(* CODESYS project tc3_utilities_extension.library
   Author: Csaba Attila Biro
   Placeholder: Tc3_Utilities_Extension
   Title: Tc3_Utilities_Extension
   Version: 2.4.92
   Company: Harman

Project tree, tasks and I/O mapping:
  libraries: Tc2_EtherCAT, * (Beckhoff Automation GmbH); Tc2_IoFunctions, * (Beckhoff Automation GmbH); Tc2_Standard, * (Beckhoff Automation GmbH); Tc2_System, * (Beckhoff Automation GmbH); Tc2_TcpIp, * (Beckhoff Automation GmbH); Tc2_Utilities, * (Beckhoff Automation GmbH); Tc3_EventLogger, * (Beckhoff Automation GmbH); Tc3_JsonXml, * (Beckhoff Automation GmbH); Tc3_Module, * (Beckhoff Automation GmbH)
  ConfigManager/
    function block FB_ConfigManager [ST]: FB_CALL_ACT, CREATE_PATH, Load, Save
  DataManager/
    JSON/
      function ANY_TO_JSON [ST]
      function CFG_TO_JSON [ST]
      global variables JSON_GVL
      function JSON_TO_ANY [ST]
      function JSON_TO_CFG [ST]
  EtherCatDiagnostic/
    DUTs/
      data type E_EcatDiagState
      data type E_EcCommState
      data type ST_EcMasterDevState
      data type ST_PortAddr
      data type ST_SlaveState
      data type ST_SlaveStateInfo
      data type ST_SlaveStateInfoScanned
      data type ST_TopologyData
    GVLs/
      global variables DIAG_GVL
    function block FB_EtherCATDiag [ST]: DiagnosticJson, M_CheckMasterDevState, M_GetScannedSlaveName, M_GetSlaveAdresses, M_GetSlaveIdentity, M_GetSlaveName, M_GetSlaveStates, M_GetTopoData, M_GetTopoDataLen, M_ScanSlaves
    function block FB_EtherCATDiagnosticWrapper [ST]
    function block FB_EtherCATFrameDiag [ST]
    function block FB_EtherCATSlaveInfo [ST]: M_GetScannedSlaveName, M_GetSlaveAdresses, M_GetSlaveIdentity, M_GetSlaveName, M_GetSlaveStates, M_GetTopoData, M_GetTopoDataLen, M_ScanSlaves
  EventLogger/
    DUTs/
      data type E_SubSystem
    global variables EVENT_GVL
    function block FB_EventHandler [ST]
    function block FB_EventLogger [ST]
  RecipeManager/
    function block FB_RecipeManager [ST]: ENUM_FILE_LIST_ACT, FB_CALL_ACT, CREATE_PATH, Load, RefreshNameList, Save, ValidateRecipe
  Tcp Barcode Reader/
    function block FB_BARCODE_READER [ST]: FB_CALL_ACT, READ, READ_REF
  TcpIpClients/
    DUTs/
      data type ENUM_DATA_EXCHANGE_STATE
    GVLs/
      global variables TCP_GVL
    function block FB_TCP_IP_CLIENT [ST]: FB_CALL_ACT, SEND
    function block FB_TCP_IP_CLIENT_LDAT [ST]: FB_CALL_ACT, SEND
  Test/
    DUTs/
      data type E_Task
      data type E_TaskState
      data type ST_Recipe
      data type ST_RecipeTask
    TASKs/
    program MAIN [ST]: FB_CALL_ACT
  TextFileHandlers/
    function block FB_ReadTextFile [ST]: Read
    function block FB_WriteTextFile [ST]: Write
    global variables FILE_GVL
  Version/
    global variables Global_Version
*)

// EtherCatDiagnostic/DUTs/E_EcatDiagState
{attribute 'to_string'}
TYPE E_EcatDiagState :
(
	Idle := 0,
    GetSlaveAddresses := 1,
    GetSlaveStates := 2,
    GetTopoDataLen := 3,
    GetTopoData := 4,
    ScanSlaves := 5,
    GetSlaveIdentity := 6,
    GetSlaveName := 7,
    GetScannedSlaveName := 8,
    LogDiagnostics := 9,
    Done := 8000
);
END_TYPE

// EtherCatDiagnostic/DUTs/E_EcCommState
TYPE E_EcCommState : (
	eEcState_UNDEFINED 	:= 0,
	eEcState_INIT 		:= 1,
	eEcState_PREOP 		:= 2,
	eEcState_BOOT 		:= 3,
	eEcState_SAFEOP 	:= 4,
	eEcState_OP 		:= 8
) UDINT;
END_TYPE

// EtherCatDiagnostic/DUTs/ST_EcMasterDevState
{attribute 'to_string'}
TYPE ST_EcMasterDevState :
STRUCT
	eEcState	 		: E_EcCommState;
	nReserved			: ARRAY [0..2] OF UINT;

	bLinkError			: BOOL;
	bResetRequired		: BOOL;
	bMissFrmRedMode		: BOOL;
	bWatchdogTriggerd	: BOOL;
	bDriverNotFound		: BOOL;
	bResetActive		: BOOL;
	bAtLeastOneNotInOp	: BOOL;
	bDcNotInSync		: BOOL;
END_STRUCT
END_TYPE

// EtherCatDiagnostic/DUTs/ST_PortAddr
{attribute 'to_string'}
TYPE ST_PortAddr :
STRUCT
	portA : UINT;
	portB : UINT;
	portC : UINT;
	portD : UINT;
END_STRUCT
END_TYPE

// EtherCatDiagnostic/DUTs/ST_SlaveState
{attribute 'to_string'}
TYPE ST_SlaveState :
STRUCT
	(* slave state *)
	eEcState 		: E_EcCommState;
	nReserved		: UINT;
	bError			: BOOL;
	bInvalidVPRS	: BOOL;
	nReserved2		: UINT;

	(* link state *)
	bNoCommToSlave	: BOOL;
	bLinkError		: BOOL;
	bMissingLink	: BOOL;
	bUnexpectedLink	: BOOL;
	bPortA			: BOOL;
	bPortB			: BOOL;
	bPortC			: BOOL;
	bPortD			: BOOL;
END_STRUCT
END_TYPE

// EtherCatDiagnostic/DUTs/ST_SlaveStateInfo
{attribute 'to_string'}
TYPE ST_SlaveStateInfo :
STRUCT
	nIndex 			: DINT;
	sName 			: STRING(255); 		(* name of slave given in System Manager *)
	sType 			: STRING(255);		(* type of slave, e.g. EK1100*)
	nECAddr 		: UINT;			(* EtherCAT Slave Addr *)
	bDiagData		: BOOL;			(* DiagData in Slave State *)
	stPortCRCErrors	: ST_EcCrcErrorEx;(* Slave CRC-Errors, separate for each Port *)
	nSumCRCErrors	: UDINT;		(* Slave CRC-Errors, sum of all Ports *)
	stState 		: ST_SlaveState;(* EtherCAT State and Link state*)
END_STRUCT
END_TYPE

// EtherCatDiagnostic/DUTs/ST_SlaveStateInfoScanned
{attribute 'to_string'}
TYPE ST_SlaveStateInfoScanned :
STRUCT
	nIndex 			: DINT;
	sName 			: STRING; 		(* name of slave given in System Manager *)
	sType 			: STRING;		(* type of slave, e.g. EK1100*)
	nECAddr 		: UINT;			(* EtherCAT Slave Addr *)
	bDifferentName	: BOOL;			(* Name of Scanned configuration differs from Configured configuration *)
	bDifferentType	: BOOL;			(* Type Of Scanned configuration differs from Configured configuration *)
	bDifferentAddr	: BOOL;			(* EcAddress of Scanned configuration differs from Configured configuration *)
END_STRUCT
END_TYPE

// EtherCatDiagnostic/DUTs/ST_TopologyData
{attribute 'to_string'}
TYPE ST_TopologyData :
STRUCT
	iOwnPhysicalAddr 	: UINT;
	iOwnAutoIncAddr		: UINT;
	stPhysicalAddr		: ST_PortAddr;
	stAutoIncAddr		: ST_PortAddr;
	iPortDelay			: ARRAY [0..2] OF UDINT; (* EC_AD, EC_DB, EC_BC *)
	iReserved			: ARRAY [0..7] OF UDINT;
END_STRUCT
END_TYPE

// EventLogger/DUTs/E_SubSystem
TYPE E_SubSystem :
(
	NILVALUE := 0,
	SAFETY := 1,
	LOGIC := 2,
	MOTION := 3,
	FIELDBUS := 4,
	PNEUMATIC := 5,
	ELECTRIC := 6
)WORD;
END_TYPE

// TcpIpClients/DUTs/ENUM_DATA_EXCHANGE_STATE
TYPE ENUM_DATA_EXCHANGE_STATE :
(
	E_IDLE := 0,
	E_SEND_START := 100,
	E_SEND_WAIT := 200,
	E_RECEIVE_START := 300,
	E_RECEIVE_WAIT := 400,
	E_DONE := 2000,
	
	E_ERROR:=15000		
);
END_TYPE

// Test/DUTs/E_Task
TYPE E_Task :
(
	TASK_START:=0,
	TASK_MOVE,
	TASK_TAKE_SCREW,
	TASK_SCREWING,
	TASK_BARCODE_SCANN,
	TASK_CAMERA_CHECK,
	TASK_ADAPTER,
	TASK_END
	
(*
	TASK_START:= 			'EMPTY'
	TASK_MOVE:=				'X:=-86.36;Y:=168.56;Z:=115.23;C:=90.12;'
	TASK_TAKE_SCREW:=		'X:=-86.36;Y:=168.56;Z:=115.23;C:=90.12;FEEDER:=2;'
	TASK_SCREWING:=			'PRE_SCREWING:=111;MAIN_SCREWING:=11;DEPTH_TARGET:=5.89;DEPTH_REF:=11.96;'
	TASK_BARCODE_SCANN:=	'IP_ADDRESS:=192.168.0.51;'
	TASK_CAMERA_CHECK:=		'PRG_ID:=192.168.0.51;',
	TASK_ADAPTER:=			'ADAPTER_TASK_ID:=2;',
	TASK_END:= 				'EMPTY'
*)

);
END_TYPE

// Test/DUTs/E_TaskState
TYPE E_TaskState :
(
	TASK_READY:=0,
	TASK_BUSY,
	TASK_DONE,
	TASK_OK,
	TASK_NG
);
END_TYPE

// Test/DUTs/ST_Recipe
TYPE ST_Recipe :
STRUCT
	DESCRIPTION:		STRING(100);
	RECIPE_LOADED:		BOOL;
	TASK_LIST:			ARRAY [1..500] OF ST_RecipeTask;	
END_STRUCT
END_TYPE

// Test/DUTs/ST_RecipeTask
TYPE ST_RecipeTask :
STRUCT
	SLOT_CHANGE:			BOOL:=FALSE;	(* Change slot after finished this position TASK *)	
	TASK:					E_Task;		(* Describe what we want to do in *)
	TASK_COMMENT:			STRING;
	TASK_PARAMETER:			STRING(255);
	
	(*
		TASK_START:= 			'EMPTY'
		TASK_MOVE:=				'X:=-86.36;Y:=168.56;Z:=115.23;C:=90.12;'
		TASK_TAKE_SCREW:=		'X:=-86.36;Y:=168.56;Z:=115.23;C:=90.12;FEEDER:=2;'
		TASK_SCREWING:=			'PRE_SCREWING:=111;MAIN_SCREWING:=11;DEPTH_TARGET:=5.89;DEPTH_REF:=11.96;'
		TASK_BARCODE_SCANN:=	'IP_ADDRESS:=192.168.0.51;'
		TASK_CAMERA_CHECK:=		'PRG_ID:=192.168.0.51;',
		TASK_ADAPTER:=			'ADAPTER_TASK_ID:=2;',
		TASK_END:= 				'EMPTY'
	*)
	
	TASK_RESULT:			E_TaskState;
END_STRUCT
END_TYPE

// DataManager/JSON/JSON_GVL
VAR_GLOBAL CONSTANT
	MAX_JSON_LENGTH:UDINT:=1000000; //1MB - 0.001GB
	CFG_JSON_LENGTH:UDINT:=15000;
END_VAR

// EtherCatDiagnostic/GVLs/DIAG_GVL
VAR_GLOBAL CONSTANT
	iSLAVEADDR_ARR_SIZE	: UINT := 256;
    ESC_MAX_PORTS : UINT := 3;
END_VAR

// EventLogger/EVENT_GVL
{attribute 'qualified_only'}
VAR_GLOBAL
	G_bAlarmActive:			BOOL;
	G_sAlarmMessage:		STRING(255);
	G_sAlarmSource:			STRING(255);
	G_sAlarmJson:			STRING(7000);
END_VAR

// TcpIpClients/GVLs/TCP_GVL
VAR_GLOBAL CONSTANT
	DEFAULT_TIMEOUT:								TIME:=T#5S;
	DEFAULT_RECONNECT:								TIME:=T#1S;
	DEFAULT_SDAT_LENGTH:							UDINT:=998;
	DEFAULT_LDAT_LENGTH:							UDINT:=49998;
	DEFAULT_STX:									BYTE:=16#02;
	DEFAULT_ETX:									BYTE:=16#03;
END_VAR

// TextFileHandlers/FILE_GVL
VAR_GLOBAL CONSTANT
	MAX_FILE_LENGTH:UDINT:=1000000; //1MB - 0.001GB
END_VAR

// Version/Global_Version
{attribute 'TcGenerated'}
{attribute 'no-analysis'}
{attribute 'linkalways'}
// This function has been automatically generated from the project information.
VAR_GLOBAL CONSTANT
	{attribute 'const_non_replaced'}
	stLibVersion_Tc3_Utilities_Extension : ST_LibVersion := (iMajor := 2, iMinor := 4, iBuild := 92, iRevision := 0, nFlags := 0, sVersion := '2.4.92');
END_VAR

// ConfigManager/FB_ConfigManager
FUNCTION_BLOCK FB_ConfigManager
VAR_INPUT
	sDef:				STRING(MAX_STRING_LENGTH):='Configuration';
	sExt:				STRING(MAX_STRING_LENGTH):='cfg';
	sFolderPath:		STRING(MAX_STRING_LENGTH):='C:\TwinCAT\Tc_Data\Configuration';
	sKey:				STRING(MAX_STRING_LENGTH):='Configuration';
	pData:				PVOID;
	nData:				UDINT;
	RESET:				BOOL;
END_VAR
VAR_OUTPUT
	READY:				BOOL;
	BUSY:				BOOL;
	DONE:				BOOL;
	
	ERROR:				BOOL;
	ERROR_ID:			UDINT;
	
	TIME_STAMP:			STRING(MAX_STRING_LENGTH);
END_VAR
VAR
	FB_SYSTIME: 		FB_LocalSystemTime:= (bEnable:= TRUE, dwCycle:= 1);
	WRITE_FILE:			FB_WriteTextFile;
	READ_FILE:			FB_ReadTextFile;
	
	JSON_STRING:		STRING(CFG_JSON_LENGTH);
	JSON_LENGTH:		UDINT;
	
	STATE:				INT;
	INIT:				BOOL:=TRUE;
	EXECUTE:			BOOL;
	
	FILE_PATH:			STRING(MAX_STRING_LENGTH);
	FILE_NAME:			STRING(MAX_STRING_LENGTH);
	RECIPE_NAME:		STRING(MAX_STRING_LENGTH):='DefaultName';
	
	FB_CreateDir: 			FB_CreateDir;
	FB_FIND_FILE: 			FB_EnumFindFileEntry:= (sNetID:= '', tTimeout:= DEFAULT_ADS_TIMEOUT);
	ENUM_FIND_FILE:			STRING(MAX_STRING_LENGTH);
	ENUM_FIND_RECIPENAME:	STRING;
	ENUM_INDEX:				UDINT:=1;
	ENUMERATE: 				BOOL;
	ENUM_STATE: 			INT;
	
	eSubSystem: 			E_SubSystem:= E_SubSystem.LOGIC;
	FB_LOGGER:				FB_EventLogger:= (eSubsystem:= eSubsystem, sJson:='{}');
END_VAR

CREATE_PATH();
FB_FIND_FILE(sPathName:= CONCAT(sFolderPath, CONCAT('\', CONCAT('*', CONCAT('.', CONCAT(sDef, CONCAT('.', sExt)))))));
FB_SYSTIME();
READY:= STATE=0;
BUSY:= STATE<>0;

IF INIT THEN
	INIT := FALSE;
	ENUMERATE:=TRUE;
    FB_CreateDir( bExecute := FALSE );
    FB_CreateDir(sNetId:= '',
                sPathName:= sFolderPath,
                ePath:= PATH_GENERIC,
                bExecute:= TRUE,
                tTimeout:= DEFAULT_ADS_TIMEOUT);
ELSE
    FB_CreateDir(bExecute := FALSE);
END_IF

CASE STATE OF
	1100:
		ENUMERATE:=TRUE;
		CREATE_PATH();
		IF CFG_TO_JSON(pData,nData, sKey:=sKey, SYSTEMTIME_TO_STRING(FB_SYSTIME.systemTime), JSON_STRING, JSON_LENGTH) THEN
			STATE:=1200;
		END_IF
	1200:
		IF WRITE_FILE.Write(FILE_PATH) THEN
			STATE:=1300;
		END_IF
	2100:
		CREATE_PATH();
		IF READ_FILE.Read(FILE_PATH) THEN
			STATE:=2200;
		END_IF
	2200:
		IF JSON_TO_CFG(pData,nData, sKey:=sKey, TIME_STAMP, JSON_STRING) THEN
			EXECUTE:=FALSE;
			ENUMERATE:=TRUE;
			STATE:=2300;
		END_IF
END_CASE

ERROR:=(ERROR_ID<>0);
FB_CALL_ACT();

ACTION FB_CALL_ACT:
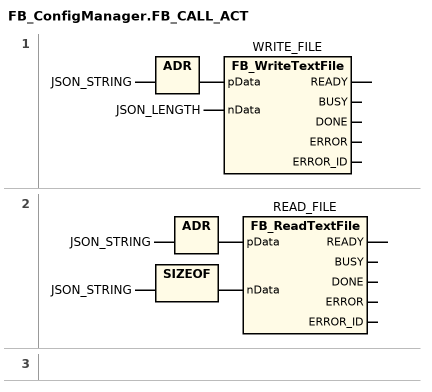
// NETWORK 1
WRITE_FILE(pData := ADR(JSON_STRING), nData := JSON_LENGTH); // FB_WriteTextFile

// NETWORK 2
READ_FILE(pData := ADR(JSON_STRING), nData := SIZEOF(JSON_STRING)); // FB_ReadTextFile

// NETWORK 3
END_ACTION

METHOD PRIVATE CREATE_PATH : BOOL
VAR_INPUT
END_VAR
FILE_NAME:=CONCAT(RECIPE_NAME, CONCAT('.', CONCAT(sDef, CONCAT('.', sExt))));
FILE_PATH:=CONCAT(sFolderPath, CONCAT('\', FILE_NAME));
END_METHOD

METHOD PUBLIC Load : BOOL
VAR_INPUT
	NAME:				STRING;
END_VAR
VAR
END_VAR
IF STATE=0 THEN
	RECIPE_NAME:=NAME;
	STATE:=2100;
END_IF

IF STATE=2300 THEN
	STATE:=0;
	Load:=TRUE;
	RETURN;
END_IF
END_METHOD

METHOD PUBLIC Save : BOOL
VAR_INPUT
	NAME:				STRING;
END_VAR
VAR
END_VAR
IF STATE=0 THEN
	RECIPE_NAME:=NAME;
	STATE:=1100;
END_IF
IF STATE=1300 THEN
	STATE:=0;
	Save:=TRUE;
	RETURN;
END_IF
END_METHOD

END_FUNCTION_BLOCK

// DataManager/JSON/CFG_TO_JSON
(*
	Convert any type to JSON string
*)
FUNCTION CFG_TO_JSON : BOOL
VAR_INPUT
	pData:					PVOID;
	nData:					UDINT;
	sKey:					STRING;
	sTimeStamp:				STRING;
	sJson:					REFERENCE TO STRING(CFG_JSON_LENGTH);
	cbJson:					REFERENCE TO UDINT;
END_VAR
VAR
	sDataType: 				STRING;
	REF_VALID:				BOOL;
	JSON_WRITER: 			FB_JsonSaxWriter;
  	JSON_DATA: 				FB_JsonReadWriteDataType;
	eSubSystem: 			E_SubSystem:= E_SubSystem.LOGIC;
	FB_LOGGER:				FB_EventLogger:= (eSubsystem:= eSubsystem);
END_VAR

REF_VALID:=(__ISVALIDREF(sJson) AND __ISVALIDREF(cbJson) AND (pData<>0 AND nData>0));

IF REF_VALID THEN
	sDataType:=JSON_DATA.GetDataTypeNameByAddress(nData:=nData, pData:=pData);
	MEMSET(ADR(sJson), 0, SIZEOF(sJson));
	JSON_WRITER.ResetDocument();
	JSON_WRITER.StartObject();
	JSON_WRITER.AddKeyString('Timestamp', sTimeStamp);
	JSON_DATA.AddJsonKeyValueFromSymbol(fbWriter:=JSON_WRITER, sKey:=sKey, sDatatype:=sDataType, nData:=nData, pData:=pData);
	JSON_WRITER.EndObject();
	cbJson:=JSON_WRITER.CopyDocument(sJson, SIZEOF(sJson));
	CFG_TO_JSON:=TRUE;
ELSE
	IF pData=0 THEN
		FB_LOGGER(sMsg:='Check data pointer failed due to invalid destination address.', eSevr:=TcEventSeverity.Error);
	ELSIF nData<=0 THEN
		FB_LOGGER(sMsg:='Check data pointer failed due to invalid size.', eSevr:=TcEventSeverity.Error);
	ELSIF NOT __ISVALIDREF(sJson) THEN
		FB_LOGGER(sMsg:='Check JSON string failed due to invalid reference.', eSevr:=TcEventSeverity.Error);
	ELSIF NOT __ISVALIDREF(cbJson) THEN
		FB_LOGGER(sMsg:='Check JSON length failed due to invalid reference.', eSevr:=TcEventSeverity.Error);
	END_IF
	CFG_TO_JSON:=TRUE;
END_IF

END_FUNCTION

// EventLogger/FB_EventLogger
{attribute 'reflection'}
FUNCTION_BLOCK FB_EventLogger
VAR_INPUT
	sMsg			: T_MaxString;
	eSevr			: TcEventSeverity	:= TcEventSeverity.Verbose;
	eSubSystem		: E_SubSystem;
	sJson			: STRING(7000)	:= '{}';
END_VAR

VAR_OUTPUT
END_VAR

VAR
	bInitialized		:	BOOL := FALSE;
	bInitFailed			:	BOOL := FALSE;
	sSubsystemSource	:	STRING;
	fbMessage			:	REFERENCE TO FB_TcMessage;
	fbAlarm				:	REFERENCE TO FB_TcAlarm;
	fbMessages 			:	ARRAY [0..4] OF FB_TcMessage;
	fbAlarms			:	ARRAY [0..4] OF FB_TcAlarm;
	fbSource 			:	FB_TcSourceInfo;
	hr 					:	HRESULT;
	hrLastInternalError :	HRESULT;
	eTraceLevel 		:	TcEventSeverity := TcEventSeverity.Verbose;
	
	{attribute 'instance-path'} 
    {attribute 'noinit'} 
	sPath				:	T_MaxString;
END_VAR

IF NOT bInitialized AND NOT bInitFailed THEN
	//Messages
	hr := fbMessages[TC_EVENTS.GeneralEventClass.Verbose.nEventId].CreateEx(TC_EVENTS.GeneralEventClass.Verbose, 0);
	IF FAILED(hr) THEN
		bInitFailed := TRUE;
		hrLastInternalError := hr;
	END_IF
	hr := fbMessages[TC_EVENTS.GeneralEventClass.Info.nEventId].CreateEx(TC_EVENTS.GeneralEventClass.Info, 0);
	IF FAILED(hr) THEN
		bInitFailed := TRUE;
		hrLastInternalError := hr;
	END_IF
	hr := fbMessages[TC_EVENTS.GeneralEventClass.Warning.nEventId].CreateEx(TC_EVENTS.GeneralEventClass.Warning, 0);
	IF FAILED(hr) THEN
		bInitFailed := TRUE;
		hrLastInternalError := hr;
	END_IF
	//Alarm messages
	hr := fbMessages[TC_EVENTS.GeneralEventClass.Error.nEventId].CreateEx(TC_EVENTS.GeneralEventClass.Error, 0);
	IF FAILED(hr) THEN
		bInitFailed := TRUE;
		hrLastInternalError := hr;
	END_IF
	hr := fbMessages[TC_EVENTS.GeneralEventClass.Critical.nEventId].CreateEx(TC_EVENTS.GeneralEventClass.Critical, 0);
	IF FAILED(hr) THEN
		bInitFailed := TRUE;
		hrLastInternalError := hr;
	END_IF	
	//Alarms
	hr := fbAlarms[TC_EVENTS.GeneralEventClass.Error.nEventId].CreateEx(TC_EVENTS.GeneralEventClass.Error, TRUE, 0);
	IF FAILED(hr) THEN
		bInitFailed := TRUE;
		hrLastInternalError := hr;
	END_IF
	hr := fbAlarms[TC_EVENTS.GeneralEventClass.Critical.nEventId].CreateEx(TC_EVENTS.GeneralEventClass.Critical, TRUE, 0);
	IF FAILED(hr) THEN
		bInitFailed := TRUE;
		hrLastInternalError := hr;
	END_IF	
	
	//Init failed
	IF bInitFailed THEN
		ADSLOGSTR(msgCtrlMask := ADSLOG_MSGTYPE_ERROR, msgFmtStr:='[LOGGER] Initialization failed in %s', strArg:=sPath); 
	ELSE
		bInitialized := TRUE;
	END_IF
END_IF
IF bInitFailed THEN
	RETURN;
END_IF
CASE eSevr OF
	//Messages
	TcEventSeverity.Verbose: 	fbMessage REF= fbMessages[TC_EVENTS.GeneralEventClass.Verbose.nEventId];
	TcEventSeverity.Info:		fbMessage REF= fbMessages[TC_EVENTS.GeneralEventClass.Info.nEventId];	
	TcEventSeverity.Warning:	fbMessage REF= fbMessages[TC_EVENTS.GeneralEventClass.Warning.nEventId];
	//Alarms
	TcEventSeverity.Error:		
		fbMessage REF= fbMessages[TC_EVENTS.GeneralEventClass.Error.nEventId]; 
		fbAlarm REF= fbAlarms[TC_EVENTS.GeneralEventClass.Error.nEventId]; 
	TcEventSeverity.Critical:	
		fbMessage REF= fbMessages[TC_EVENTS.GeneralEventClass.Critical.nEventId];
		fbAlarm REF= fbAlarms[TC_EVENTS.GeneralEventClass.Critical.nEventId];
	ELSE
		RETURN;
END_CASE
CASE eSubsystem OF
	E_Subsystem.FIELDBUS: sSubsystemSource := ' - EtherCAT';
	E_Subsystem.MOTION: sSubsystemSource := ' - Motion';
	E_Subsystem.SAFETY: sSubsystemSource := ' - Safety';
	E_Subsystem.LOGIC: sSubsystemSource := ' - Logic';
	E_Subsystem.PNEUMATIC: sSubsystemSource := ' - Pneumatic';	
	E_Subsystem.ELECTRIC: sSubsystemSource := ' - Electric';	
	ELSE
		sSubsystemSource := 'Unknown';
END_CASE
sMsg:=CONCAT(' ',CONCAT(sMsg,' '));
IF eSevr=TcEventSeverity.Verbose OR eSevr=TcEventSeverity.Info OR eSevr=TcEventSeverity.Warning THEN
	fbSource.sName :=CONCAT(sPath, sSubsystemSource);
	hr := fbMessage.CreateEx(stEventEntry:=fbMessage.stEventEntry, ipSourceInfo:=fbSource);
	fbMessage.ipArguments.Clear();
	fbMessage.ipArguments.AddString(sMsg);
	IF LEN(sJson) = 0 THEN
		sJson := '{}';
	END_IF
	fbMessage.SetJsonAttribute(sJson);
	IF NOT FAILED(hr) AND fbMessage.eSeverity >= eTraceLevel THEN
		hr := fbMessage.Send(0);
	END_IF
	IF FAILED(hr) THEN
		hrLastInternalError := hr;
	END_IF
ELSIF eSevr=TcEventSeverity.Error OR eSevr=TcEventSeverity.Critical THEN
	fbSource.sName :=CONCAT(sPath, sSubsystemSource);
	hr := fbAlarm.CreateEx(stEventEntry:=fbAlarm.stEventEntry, ipSourceInfo:=fbSource, bWithConfirmation:=TRUE);
	fbAlarm.ipArguments.Clear();
	
	fbAlarm.ipArguments.AddString(sMsg);
	IF LEN(sJson) = 0 THEN
		sJson := '{}';
	END_IF
	fbAlarm.SetJsonAttribute(sJson);
	IF NOT FAILED(hr) AND fbAlarm.eSeverity >= eTraceLevel THEN
		hr := fbAlarm.Raise(0);
		EVENT_GVL.G_sAlarmJson:=sJson;
		EVENT_GVL.G_sAlarmSource:=fbSource.sName;
		EVENT_GVL.G_sAlarmMessage:=sMsg;
		EVENT_GVL.G_bAlarmActive:=TRUE;
	END_IF
	IF FAILED(hr) THEN
		hrLastInternalError := hr;
	END_IF
	hr := fbMessage.CreateEx(stEventEntry:=fbMessage.stEventEntry, ipSourceInfo:=fbSource);
	fbMessage.ipArguments.Clear();
	fbMessage.ipArguments.AddString(sMsg);
	IF LEN(sJson) = 0 THEN
		sJson := '{}';
	END_IF
	fbMessage.SetJsonAttribute(sJson);
	IF NOT FAILED(hr) AND fbMessage.eSeverity >= eTraceLevel THEN
		hr := fbMessage.Send(0);
	END_IF
	IF FAILED(hr) THEN
		hrLastInternalError := hr;
	END_IF
END_IF

END_FUNCTION_BLOCK

// DataManager/JSON/JSON_TO_CFG
(*
	Convert JSON string to any sutitable type
*)
FUNCTION JSON_TO_CFG : BOOL
VAR_INPUT
	pData:					PVOID;
	nData:					UDINT;
	sKey:					STRING;
	sTimeStamp:				REFERENCE TO STRING;
	sJson:					REFERENCE TO STRING(CFG_JSON_LENGTH);
END_VAR
VAR
	sDataType: 				STRING;
	sDataSymbol:			STRING;
	REF_VALID:				BOOL;
	JSON_DOM_PARSER: 		FB_JsonDomParser;
	JSON_DOC: 				SJsonValue;
	JSON_TIME: 				SJsonValue;
	JSON_CONTENT:			SJsonValue;
  	JSON_DATA: 				FB_JsonReadWriteDataType;
	eSubSystem: 			E_SubSystem:= E_SubSystem.LOGIC;
	FB_LOGGER:				FB_EventLogger:= (eSubsystem:= eSubsystem);
END_VAR

REF_VALID:=(__ISVALIDREF(sJson) AND __ISVALIDREF(sTimeStamp) AND (pData<>0 AND nData>0));

IF REF_VALID THEN
	sDataType:=JSON_DATA.GetDataTypeNameByAddress(nData:=nData, pData:=pData);
	sDataSymbol:=JSON_DATA.GetSymbolNameByAddress(nData:=nData, pData:=pData);
	
	JSON_DOC:=JSON_DOM_PARSER.ParseDocument(sJson);
	IF JSON_DOM_PARSER.HasMember(JSON_DOC, 'Timestamp') THEN
		JSON_TIME:=JSON_DOM_PARSER.FindMember(JSON_DOC, 'Timestamp');
		sTimeStamp:=JSON_DOM_PARSER.GetString(JSON_TIME);
	END_IF
	IF JSON_DOM_PARSER.HasMember(JSON_DOC, sKey) THEN
		MEMSET(ADR(sJson), 0, SIZEOF(sJson));
		JSON_CONTENT:=JSON_DOM_PARSER.FindMember(JSON_DOC, sKey);
		JSON_DOM_PARSER.CopyJson (JSON_CONTENT, sJson, SIZEOF(sJson));
		JSON_DATA.SetSymbolFromJson(sJson:=sJson, sDatatype:=sDataType, nData:=nData, pData:=pData);
	END_IF
	JSON_TO_CFG:=TRUE;
ELSE
	IF pData=0 THEN
		FB_LOGGER(sMsg:='Check data pointer failed due to invalid destination address.', eSevr:=TcEventSeverity.Error);
	ELSIF nData<=0 THEN
		FB_LOGGER(sMsg:='Check data pointer failed due to invalid size.', eSevr:=TcEventSeverity.Error);
	ELSIF NOT __ISVALIDREF(sJson) THEN
		FB_LOGGER(sMsg:='Check JSON string failed due to invalid reference.', eSevr:=TcEventSeverity.Error);
	ELSIF NOT __ISVALIDREF(sTimeStamp) THEN
		FB_LOGGER(sMsg:='Check TimeStamp string failed due to invalid reference.', eSevr:=TcEventSeverity.Error);
	END_IF
	JSON_TO_CFG:=TRUE;
END_IF

END_FUNCTION

// TextFileHandlers/FB_WriteTextFile
{attribute 'reflection'}
FUNCTION_BLOCK FB_WriteTextFile
VAR_INPUT
	pData:				PVOID;
	nData:				UDINT;
END_VAR
VAR_OUTPUT
	READY:				BOOL;
	BUSY:				BOOL;
	DONE:				BOOL;
	ERROR:				BOOL;
	ERROR_ID:			UDINT;
END_VAR
VAR
	FB_FileWrite:		FB_FileWrite;
	FB_FileOpen:		FB_FileOpen;
	FB_FileClose:		FB_FileClose;
	sPath:				STRING(MAX_STRING_LENGTH);
	H_DEST_FILE:		UINT:= 0;
	STATE:				INT;
	EXECUTE:			BOOL;
	
	eSubSystem: 			E_SubSystem:= E_SubSystem.LOGIC;
	FB_LOGGER:				FB_EventLogger:= (eSubsystem:= eSubsystem);
END_VAR

READY:= STATE=0;
BUSY:= STATE<>0;
CASE STATE OF
	0:
		IF EXECUTE THEN
			ERROR_ID:=0;
			DONE:=FALSE;
			STATE:=100;
		END_IF
	100:
		FB_FileOpen( bExecute := FALSE );
		FB_FileOpen( sNetId := '', sPathName := sPath,
					 nMode := FOPEN_MODEWRITE OR FOPEN_MODETEXT,
					 ePath := PATH_GENERIC, tTimeout := DEFAULT_ADS_TIMEOUT, bExecute := TRUE );
		STATE:=200;
    200:
		FB_FileOpen( bExecute := FALSE );
		IF NOT FB_FileOpen.bBusy THEN
			IF FB_FileOpen.bError THEN
				ERROR_ID:=FB_FileOpen.nErrId;
				FB_LOGGER(sMsg:=CONCAT('FB_FileOpen throw an error: ', DWORD_TO_HEXSTR(ERROR_ID, 0, FALSE )), eSevr:=TcEventSeverity.Error);
				STATE:=700;
			ELSE
				H_DEST_FILE := FB_FileOpen.hFile;
				STATE:=300;
			END_IF
		END_IF
	300:
		FB_FileWrite( bExecute := FALSE );
        FB_FileWrite( sNetId:='', 
					  hFile:=H_DEST_FILE,
                      pWriteBuff:= pData, 
					  cbWriteLen:= (nData-1),
                      bExecute:=TRUE, 
					  tTimeout:=DEFAULT_ADS_TIMEOUT );
		STATE:=400;
	400:
		FB_FileWrite( bExecute := FALSE );
		IF NOT FB_FileWrite.bBusy THEN
			IF FB_FileWrite.bError THEN
				ERROR_ID:=FB_FileWrite.nErrId;
				FB_LOGGER(sMsg:=CONCAT('FB_FileWrite throw an error: ', DWORD_TO_HEXSTR(ERROR_ID, 0, FALSE )), eSevr:=TcEventSeverity.Error);
				STATE:=700;
			ELSE
				STATE:=500;
			END_IF
		END_IF
	 500:
         FB_FileClose( bExecute := FALSE );
         FB_FileClose( sNetId:='', hFile:=H_DEST_FILE, bExecute:=TRUE, tTimeout:=DEFAULT_ADS_TIMEOUT );
         STATE:=600;
     600:
		FB_FileClose( bExecute := FALSE );
		IF NOT FB_FileClose.bBusy THEN
			IF FB_FileClose.bError THEN
				ERROR_ID:=FB_FileClose.nErrId;
				FB_LOGGER(sMsg:=CONCAT('FB_FileClose throw an error: ', DWORD_TO_HEXSTR(ERROR_ID, 0, FALSE )), eSevr:=TcEventSeverity.Error);
			END_IF
			STATE:=700;
			DONE:=TRUE;
			H_DEST_FILE:= 0;
		END_IF
	700:
		IF NOT EXECUTE THEN
			STATE:=0;
		END_IF
END_CASE

METHOD PUBLIC Write : BOOL
VAR_INPUT
	sFilePath:		STRING(MAX_STRING_LENGTH);
END_VAR
IF sFilePath<>'' THEN
	IF STATE=700 THEN
		EXECUTE:=FALSE;
		Write:=TRUE;
	END_IF
	
	IF STATE=0 THEN
		sPath:=sFilePath;
		EXECUTE:=TRUE;
	END_IF	
END_IF
END_METHOD

END_FUNCTION_BLOCK

// TextFileHandlers/FB_ReadTextFile
{attribute 'reflection'}
FUNCTION_BLOCK FB_ReadTextFile
VAR_INPUT
	pData:				PVOID;
	nData:				UDINT;
END_VAR
VAR_OUTPUT
	READY:				BOOL;
	BUSY:				BOOL;
	DONE:				BOOL;
	ERROR:				BOOL;
	ERROR_ID:			UDINT;
END_VAR
VAR
	FB_FileRead:		FB_FileRead;
	FB_FileOpen:		FB_FileOpen;
	FB_FileClose:		FB_FileClose;
	sPath:				STRING(MAX_STRING_LENGTH);
	H_SCR_FILE:			UINT:= 0;
	STATE:				INT;
	EXECUTE:			BOOL;
	
	eSubSystem: 			E_SubSystem:= E_SubSystem.LOGIC;
	FB_LOGGER:				FB_EventLogger:= (eSubsystem:= eSubsystem);
END_VAR

READY:= STATE=0;
BUSY:= STATE<>0;
CASE STATE OF
	0:
		IF EXECUTE THEN
			ERROR_ID:=0;
			DONE:=FALSE;
			MEMSET(pData, 0, nData);
			STATE:=100;
		END_IF
	100:	
		FB_FileOpen( bExecute := FALSE );
		FB_FileOpen( sNetId := '', sPathName := sPath,
					 nMode := FOPEN_MODEREAD OR FOPEN_MODETEXT,
					 ePath := PATH_GENERIC, tTimeout := DEFAULT_ADS_TIMEOUT, bExecute := TRUE );
		STATE:=200;
	200:
		FB_FileOpen( bExecute := FALSE );
		IF NOT FB_FileOpen.bBusy THEN
			IF FB_FileOpen.bError THEN
				ERROR_ID:=FB_FileOpen.nErrId;
				FB_LOGGER(sMsg:=CONCAT(CONCAT('FB_FileOpen throw an error: ', DWORD_TO_HEXSTR(ERROR_ID, 0, FALSE )),CONCAT(' Path: ', sPath)), eSevr:=TcEventSeverity.Error);
				STATE:=700;
			ELSE
				H_SCR_FILE := FB_FileOpen.hFile;
				STATE:=300;
			END_IF
		END_IF
	300:
		FB_FileRead( bExecute:= FALSE );
		FB_FileRead( sNetId:='', hFile:=H_SCR_FILE,
					pReadBuff:= pData, cbReadLen:= nData,
					bExecute:=TRUE, tTimeout:=DEFAULT_ADS_TIMEOUT);
		STATE:=400;
	400:
		FB_FileRead( bExecute:= FALSE );
		IF NOT FB_FileRead.bBusy THEN
			IF FB_FileRead.bError THEN
				ERROR_ID:=FB_FileRead.nErrId;
				FB_LOGGER(sMsg:=CONCAT('FB_FileRead throw an error: ', DWORD_TO_HEXSTR(ERROR_ID, 0, FALSE )), eSevr:=TcEventSeverity.Error);
				STATE:=700;
			ELSE
				STATE:=500;
			END_IF
		END_IF
	500:
         FB_FileClose( bExecute := FALSE );
         FB_FileClose( sNetId:='', hFile:=H_SCR_FILE, bExecute:=TRUE, tTimeout:=DEFAULT_ADS_TIMEOUT );
         STATE:=600;
	600:
		FB_FileClose( bExecute := FALSE );
		IF NOT FB_FileClose.bBusy THEN
			IF FB_FileClose.bError THEN
				ERROR_ID:=FB_FileClose.nErrId;
				FB_LOGGER(sMsg:=CONCAT('FB_FileClose throw an error: ', DWORD_TO_HEXSTR(ERROR_ID, 0, FALSE )), eSevr:=TcEventSeverity.Error);
			END_IF
			STATE:=700;
			DONE:=TRUE;
			H_SCR_FILE := 0;
		END_IF
	700:
		IF NOT EXECUTE THEN
			STATE:=0;
		END_IF
END_CASE

ERROR:=(ERROR_ID<>0);

METHOD PUBLIC Read : BOOL
VAR_INPUT
	sFilePath:		STRING(MAX_STRING_LENGTH);
END_VAR
IF sFilePath<>'' THEN
	IF STATE=700 THEN
		EXECUTE:=FALSE;
		Read:=TRUE;
	END_IF
	
	IF STATE=0 THEN
		sPath:=sFilePath;
		EXECUTE:=TRUE;
	END_IF
END_IF
END_METHOD

END_FUNCTION_BLOCK

// DataManager/JSON/ANY_TO_JSON
(*
	Convert any type to JSON string
*)
FUNCTION ANY_TO_JSON : BOOL
VAR_INPUT
	pData:					PVOID;
	nData:					UDINT;
	sKey:					STRING;
	sTimeStamp:				STRING;
	sJson:					REFERENCE TO STRING(MAX_JSON_LENGTH);
	cbJson:					REFERENCE TO UDINT;
END_VAR
VAR
	sDataType: 				STRING;
	REF_VALID:				BOOL;
	JSON_WRITER: 			FB_JsonSaxWriter;
  	JSON_DATA: 				FB_JsonReadWriteDataType;
	eSubSystem: 			E_SubSystem:= E_SubSystem.LOGIC;
	FB_LOGGER:				FB_EventLogger:= (eSubsystem:= eSubsystem);
END_VAR

REF_VALID:=(__ISVALIDREF(sJson) AND __ISVALIDREF(cbJson) AND (pData<>0 AND nData>0));

IF REF_VALID THEN
	sDataType:=JSON_DATA.GetDataTypeNameByAddress(nData:=nData, pData:=pData);
	MEMSET(ADR(sJson), 0, SIZEOF(sJson));
	JSON_WRITER.ResetDocument();
	JSON_WRITER.StartObject();
	JSON_WRITER.AddKeyString('Timestamp', sTimeStamp);
	JSON_DATA.AddJsonKeyValueFromSymbol(fbWriter:=JSON_WRITER, sKey:=sKey, sDatatype:=sDataType, nData:=nData, pData:=pData);
	JSON_WRITER.EndObject();
	cbJson:=JSON_WRITER.CopyDocument(sJson, SIZEOF(sJson));
	ANY_TO_JSON:=TRUE;
ELSE
	IF pData=0 THEN
		FB_LOGGER(sMsg:='Check data pointer failed due to invalid destination address.', eSevr:=TcEventSeverity.Error);
	ELSIF nData<=0 THEN
		FB_LOGGER(sMsg:='Check data pointer failed due to invalid size.', eSevr:=TcEventSeverity.Error);
	ELSIF NOT __ISVALIDREF(sJson) THEN
		FB_LOGGER(sMsg:='Check JSON string failed due to invalid reference.', eSevr:=TcEventSeverity.Error);
	ELSIF NOT __ISVALIDREF(cbJson) THEN
		FB_LOGGER(sMsg:='Check JSON length failed due to invalid reference.', eSevr:=TcEventSeverity.Error);
	END_IF
	ANY_TO_JSON:=TRUE;
END_IF

END_FUNCTION

// DataManager/JSON/JSON_TO_ANY
(*
	Convert JSON string to any sutitable type
*)
FUNCTION JSON_TO_ANY : BOOL
VAR_INPUT
	pData:					PVOID;
	nData:					UDINT;
	sKey:					STRING;
	sTimeStamp:				REFERENCE TO STRING;
	sJson:					REFERENCE TO STRING(MAX_JSON_LENGTH);
END_VAR
VAR
	sDataType: 				STRING;
	sDataSymbol:			STRING;
	REF_VALID:				BOOL;
	JSON_DOM_PARSER: 		FB_JsonDomParser;
	JSON_DOC: 				SJsonValue;
	JSON_TIME: 				SJsonValue;
	JSON_CONTENT:			SJsonValue;
  	JSON_DATA: 				FB_JsonReadWriteDataType;
	eSubSystem: 			E_SubSystem:= E_SubSystem.LOGIC;
	FB_LOGGER:				FB_EventLogger:= (eSubsystem:= eSubsystem);
END_VAR

REF_VALID:=(__ISVALIDREF(sJson) AND __ISVALIDREF(sTimeStamp) AND (pData<>0 AND nData>0));

IF REF_VALID THEN
	sDataType:=JSON_DATA.GetDataTypeNameByAddress(nData:=nData, pData:=pData);
	sDataSymbol:=JSON_DATA.GetSymbolNameByAddress(nData:=nData, pData:=pData);
	JSON_DOC:=JSON_DOM_PARSER.ParseDocument(sJson);
	IF JSON_DOM_PARSER.HasMember(JSON_DOC, 'Timestamp') THEN
		JSON_TIME:=JSON_DOM_PARSER.FindMember(JSON_DOC, 'Timestamp');
		sTimeStamp:=JSON_DOM_PARSER.GetString(JSON_TIME);
	END_IF
	IF JSON_DOM_PARSER.HasMember(JSON_DOC, sKey) THEN
		MEMSET(ADR(sJson), 0, SIZEOF(sJson));
		JSON_CONTENT:=JSON_DOM_PARSER.FindMember(JSON_DOC, sKey);
		JSON_DOM_PARSER.CopyJson (JSON_CONTENT, sJson, SIZEOF(sJson));
		JSON_DATA.SetSymbolFromJson(sJson:=sJson, sDatatype:=sDataType, nData:=nData, pData:=pData);
	END_IF
	JSON_TO_ANY:=TRUE;
ELSE
	IF pData=0 THEN
		FB_LOGGER(sMsg:='Check data pointer failed due to invalid destination address.', eSevr:=TcEventSeverity.Error);
	ELSIF nData<=0 THEN
		FB_LOGGER(sMsg:='Check data pointer failed due to invalid size.', eSevr:=TcEventSeverity.Error);
	ELSIF NOT __ISVALIDREF(sJson) THEN
		FB_LOGGER(sMsg:='Check JSON string failed due to invalid reference.', eSevr:=TcEventSeverity.Error);
	ELSIF NOT __ISVALIDREF(sTimeStamp) THEN
		FB_LOGGER(sMsg:='Check TimeStamp string failed due to invalid reference.', eSevr:=TcEventSeverity.Error);
	END_IF
	JSON_TO_ANY:=TRUE;
END_IF

END_FUNCTION

// EtherCatDiagnostic/FB_EtherCATDiag
FUNCTION_BLOCK FB_EtherCATDiag
VAR_INPUT
	sIPCNetID					: T_AmsNetId; 	// AmsNetId of the IPC 
	sMasterNetID				: T_AmsNetId; 	// AmsNetId of the EtherCAT master device 
	nMasterDevID				: UINT;			// Device ID of EtherCAT master
	nSlaveCount 				: UINT;			// current slave count
	nSlaveCountCfg 				: UINT;			// configured slave count
	nMasterDevState				: WORD;			// device state of EtherCAT Master
	bAllFrameWcStatesOK			: BOOL;			// all FrameWcState OK?
	tTimeout					: TIME := T#5S; // ads timeout
    eSubSystem 					: E_SubSystem := E_SubSystem.FIELDBUS;
END_VAR
VAR_OUTPUT
	bEtherCATOK					: BOOL;			// no problem on EtherCAT
	bFrameWcStateError			: BOOL;			// error in at least one frame
	bSlaveCountError			: BOOL;			// EtherCAT slave count mismatch (# of cfg slaves <> # of found slaves)
	bMasterDevStateError		: BOOL;			// error in master device state
	stMasterDevState			: ST_EcMasterDevState; // splitted master device state
	bBusy						: BOOL;			// FB busy
	bError						: BOOL;			// FB with error
	iErrorID					: UDINT;		// FB error ID
END_VAR
VAR_IN_OUT
	arrDiagSlaveInfo 			: ARRAY [0..ESC_MAX_PORTS] OF ST_SlaveStateInfo;		// read in info from configured slaves
	arrDiagSlaveInfoScanned		: ARRAY [0..ESC_MAX_PORTS] OF ST_SlaveStateInfoScanned;	// read in info from scanned slaves
END_VAR
VAR
	sMasterOpState				: STRING(255);
	sSlaveOpState				: STRING(255);
	iState						: E_EcatDiagState;
	nMasterDevStatePrev			: WORD;
	bSlaveCountErrorPrev		: BOOL;
	bAllFrameWcStatesOKPrev		: BOOL;
	bDiagReq					: BOOL := TRUE;
	I							: UDINT;
    P							: UDINT;   
    arrSlaveInfo 				: ARRAY [0..iSLAVEADDR_ARR_SIZE] OF ST_SlaveStateInfo;
    rSlaveInfo  				: REFERENCE TO ST_SlaveStateInfo;

	(* -- Get Slave Addresses *)
	fbGetSlaveAddresses 		: FB_EcGetAllSlaveAddr;
	arrSlaveAddresses 			: ARRAY[0..iSLAVEADDR_ARR_SIZE] OF UINT;
	iNumOfSlavesRead			: UINT;

	(* -- Get Slave States *)
	fbGetAllSlaveStates			: FB_EcGetAllSlaveStates;
	arrSlaveStates 				: ARRAY[0..iSLAVEADDR_ARR_SIZE] OF ST_EcSlaveState;

	(* -- Get Topology Data *)
	iTopologyData				: UDINT;
	fbGetTopologyData			: ADSREAD;
	arrTopologyData				: ARRAY[0..iSLAVEADDR_ARR_SIZE] OF ST_TopologyData;

	(* -- Check Topology *)
	aiDiagIndex					: ARRAY [0..ESC_MAX_PORTS] OF UINT;
    iDiagIndex 					: UINT;    
	aiDiagPort					: ARRAY [0..ESC_MAX_PORTS] OF UINT;
    iDiagPort 					: UINT;
	iIdx						: DINT;

	(* -- Scan Slaves *)
	fbEcGetScannedSlaves		: FB_EcGetScannedSlaves;
	arrScannedSlaveInfo			: ARRAY [0..iSLAVEADDR_ARR_SIZE] OF ST_EcSlaveScannedData; // what...
    rScannedSlaveInfo   		: REFERENCE TO ST_EcSlaveScannedData;
	nScannedSlaves				: UINT;

	(* -- Get Slave Identities *)
	fbGetSlaveIdentity			: FB_EcGetSlaveIdentity;
	stIdentity 					: ST_EcSlaveIdentity;

	(* -- Get Slave Names *)
	fbGetSlaveName 				: IOF_GetBoxNameByAddr;
    arrSlaveInfoScanned			: ARRAY [0..iSLAVEADDR_ARR_SIZE] OF ST_SlaveStateInfoScanned; // the F
    rSlaveInfoScanned   		: REFERENCE TO ST_SlaveStateInfoScanned;
	strName						: STRING;

    // Logging components
    fbLogger 					: FB_EventLogger := (eSubsystem := eSubsystem);  
    fbJson 						: FB_JsonSaxWriter;
    fbJsonDataType 				: FB_JsonReadWriteDataType;
    rDiagSlaveInfo 				: REFERENCE TO ST_SlaveStateInfo;
    tEtherCATOK 				: F_TRIG;
    tFrameWcStateError 			: R_TRIG;
    tMasterError 				: R_TRIG;
    jsonIdx 					: UINT;
    test 						: T_MaxString;
END_VAR


(* cyclic diag *)
bFrameWcStateError := NOT bAllFrameWcStatesOK;

bSlaveCountError := (nSlaveCount <> nSlaveCountCfg) OR (nSlaveCount = 0);
IF (bSlaveCountError AND NOT bSlaveCountErrorPrev) OR (NOT bSlaveCountError AND bSlaveCountErrorPrev) THEN
	bSlaveCountErrorPrev := bSlaveCountError;
	bDiagReq := TRUE; // slave count error change detected --> diag required
END_IF

IF (bAllFrameWcStatesOK AND NOT bAllFrameWcStatesOKPrev) OR (NOT bAllFrameWcStatesOK AND bAllFrameWcStatesOKPrev) THEN
	bAllFrameWcStatesOKPrev := bAllFrameWcStatesOK;
	bDiagReq := TRUE; // frame error change detected --> diag required
END_IF

IF (nMasterDevState <> nMasterDevStatePrev) THEN
	M_CheckMasterDevState();
	bDiagReq := TRUE; // devstate change detected --> diag required
END_IF

(* acyclic diag *)
CASE iState OF
E_EcatDiagState.Idle: (* IDLE *)
	IF bDiagReq THEN				// diag requested
		bDiagReq := FALSE;

		IF sMasterNetID <> '' AND sMasterNetID <> '0.0.0.0.0.0' THEN
			iState := E_EcatDiagState.GetSlaveAddresses;	// execute diag
			bBusy := TRUE;
		ELSE
			bError := TRUE;
			iErrorID := 7;
		END_IF

		bEtherCATOK := FALSE;
	ELSE
		// check for changes in idle
		IF (bSlaveCountError OR bMasterDevStateError OR NOT bAllFrameWcStatesOK) AND NOT (arrSlaveInfo[aiDiagIndex[0]].bDiagData) THEN
			bEtherCATOK := FALSE;
			bDiagReq := TRUE;//new error --> diag requested    
		ELSIF (bSlaveCountError AND NOT bSlaveCountErrorPrev) OR (NOT bSlaveCountError AND bSlaveCountErrorPrev) THEN
			bSlaveCountErrorPrev := bSlaveCountError;
			bEtherCATOK := FALSE;
			bDiagReq := TRUE;// slave count error change detected --> diag required
		ELSIF (nMasterDevState <> nMasterDevStatePrev) THEN
			bEtherCATOK := FALSE;
			bDiagReq := TRUE;// devstate change detected --> diag required
		ELSIF (bAllFrameWcStatesOK AND NOT bAllFrameWcStatesOKPrev) OR (NOT bAllFrameWcStatesOK AND bAllFrameWcStatesOKPrev) THEN
			bAllFrameWcStatesOKPrev := bAllFrameWcStatesOK;
			bEtherCATOK := FALSE;
			bDiagReq := TRUE;// frame error change detected --> diag required
		ELSIF (bSlaveCountError OR bMasterDevStateError OR NOT bAllFrameWcStatesOK OR arrSlaveInfo[aiDiagIndex[0]].bDiagData) THEN
			bEtherCATOK := FALSE;
		ELSE
			bEtherCATOK := TRUE;
		END_IF
	END_IF

E_EcatDiagState.GetSlaveAddresses: (* get adresses *)
	M_GetSlaveAdresses();

E_EcatDiagState.GetSlaveStates: (* get states *)
	M_GetSlaveStates();

E_EcatDiagState.GetTopoDataLen:	(* get topology data length *)
	M_GetTopoDataLen();

E_EcatDiagState.GetTopoData:	(* get topology data *)
	M_GetTopoData();

E_EcatDiagState.ScanSlaves:	(* scan slaves *)
	M_ScanSlaves();

E_EcatDiagState.GetSlaveIdentity:	(* get identity *)
	M_GetSlaveIdentity();

E_EcatDiagState.GetSlaveName:	(* get name *)
	M_GetSlaveName();

E_EcatDiagState.GetScannedSlaveName:	(* get scanned name *)
	M_GetScannedSlaveName();

E_EcatDiagState.LogDiagnostics: (* Log diagnostics *)
    IF jsonIdx < iNumOfSlavesRead THEN // the last entry is always blank
        jsonIdx := MIN(iSLAVEADDR_ARR_SIZE, jsonIdx);
        rDiagSlaveInfo REF= arrSlaveInfo[jsonIdx];
		DiagnosticJson();
		IF rDiagSlaveInfo.sName <> '' THEN
			fbLogger(sMsg:=CONCAT('EtherCAT diagnostic result of ', rDiagSlaveInfo.sName), eSevr:=TcEventSeverity.Info);
		END_IF
        jsonIdx := jsonIdx + 1;
    ELSE
        jsonIdx := 0;
        iState := E_EcatDiagState.Done;    
	END_IF   
    
E_EcatDiagState.Done:	(* DONE *)
	bBusy := FALSE;
	iState := 0;

END_CASE

// Log messages
tEtherCATOK(CLK:=bEtherCATOK);
IF tEtherCATOK.Q THEN
    fbLogger(sMsg:='EtherCAT failure detected, starting diagnostic sequnce', eSevr:=TcEventSeverity.Critical, sJson:='');
END_IF

tFrameWcStateError(CLK:=bFrameWcStateError);
IF tFrameWcStateError.Q THEN
    fbLogger(sMsg:='WorkingCounterFrame error in at least one frame.', eSevr:=TcEventSeverity.Error, sJson:='');
END_IF

tMasterError(CLK:=bMasterDevStateError);
IF tMasterError.Q THEN
	CASE stMasterDevState.eEcState OF
		0: sMasterOpState:= 'UNDEFINED';
		1: sMasterOpState:= 'INIT';
		2: sMasterOpState:= 'PREOP';
		3: sMasterOpState:= 'BOOT';
		4: sMasterOpState:= 'SAFEOP';
		8: sMasterOpState:= 'OP';
	END_CASE
    fbJson.StartObject();
        fbJson.AddKey('EtherCAT Master Diagnostic');
        fbJson.StartObject();
            fbJson.AddKey('At least one not in OP state');
            fbJson.AddBool(stMasterDevState.bAtLeastOneNotInOp);
            fbJson.AddKey('DC not in sync');
            fbJson.AddBool(stMasterDevState.bDcNotInSync);
            fbJson.AddKey('Driver not found');
            fbJson.AddBool(stMasterDevState.bDriverNotFound);
            fbJson.AddKey('Link error');
            fbJson.AddBool(stMasterDevState.bLinkError);
            fbJson.AddKey('Miss Frm red mode');
            fbJson.AddBool(stMasterDevState.bMissFrmRedMode);
            fbJson.AddKey('Reset active');
            fbJson.AddBool(stMasterDevState.bResetActive);
            fbJson.AddKey('Reset required');
            fbJson.AddBool(stMasterDevState.bResetRequired);
            fbJson.AddKey('Watchdog triggerd');
            fbJson.AddBool(stMasterDevState.bWatchdogTriggerd);
            fbJson.AddKey('EtherCAT-State');
            fbJson.AddString(sMasterOpState);
        fbJson.EndObject();
    fbJson.EndObject();
    fbJson.CopyDocument(fbLogger.sJson, SIZEOF(fbLogger.sJson));

    fbLogger(sMsg:=CONCAT('Error in EtherCAT Master device state. EtherCAT-State: ', sMasterOpState), eSevr:=TcEventSeverity.Critical);
    fbJson.ResetDocument();
END_IF

ACTION DiagnosticJson:
CASE rDiagSlaveInfo.stState.eEcState OF
	0: sSlaveOpState:= 'UNDEFINED';
	1: sSlaveOpState:= 'INIT';
	2: sSlaveOpState:= 'PREOP';
	3: sSlaveOpState:= 'BOOT';
	4: sSlaveOpState:= 'SAFEOP';
	8: sSlaveOpState:= 'OP';
END_CASE
fbJson.StartObject();
    fbJson.AddKey('EtherCAT Diagnostic');
    fbJson.StartObject();
        
        fbJson.AddKey('EtherCAT address');
        fbJson.AddUdint(rDiagSlaveInfo.nECAddr);
        
        fbJson.AddKey('Index');
        fbJson.AddDint(rDiagSlaveInfo.nIndex);
        
        fbJson.AddKey('Name');
        fbJson.AddString(rDiagSlaveInfo.sName);
        
        fbJson.AddKey('Type');
        fbJson.AddString(rDiagSlaveInfo.sType);
    
        fbJson.AddKey('Diagnostic data');
        fbJson.AddBool(rDiagSlaveInfo.bDiagData);
        
        fbJson.AddKey('EtherCAT port CRC errors');
        fbjson.StartObject();
        
            fbJson.AddKey('Port - A');
            fbJson.AddUdint(rDiagSlaveInfo.stPortCRCErrors.portA);
            fbJson.AddKey('Port - B');
            fbJson.AddUdint(rDiagSlaveInfo.stPortCRCErrors.portB);
            fbJson.AddKey('Port - C');
            fbJson.AddUdint(rDiagSlaveInfo.stPortCRCErrors.portC);
            fbJson.AddKey('Port - D');
            fbJson.AddUdint(rDiagSlaveInfo.stPortCRCErrors.portD);
            
        fbJson.EndObject();
        
        fbJson.AddKey('Summary of CRC errors');
        fbjson.AddUdint(rDiagSlaveInfo.nSumCRCErrors);
        
        fbJson.AddKey('Terminal state');
        fbJson.StartObject();
        
            fbJson.AddKey('EtherCAT-State');
            fbJson.AddString(sSlaveOpState);
//            fbJson.AddKey('Reserved 1');
//            fbJson.AddUdint(rDiagSlaveInfo.stState.nReserved);
            fbJson.AddKey('Error');
            fbJson.AddBool(rDiagSlaveInfo.stState.bError);
            fbJson.AddKey('Invalid VPRS');
            fbJson.AddBool(rDiagSlaveInfo.stState.bInvalidVPRS);
//            fbJson.AddKey('Reserved 2');
//            fbJson.AddUdint(rDiagSlaveInfo.stState.nReserved2);
            fbJson.AddKey('No communication to slave');
            fbJson.AddBool(rDiagSlaveInfo.stState.bNoCommToSlave);
            fbJson.AddKey('Link error');
            fbJson.AddBool(rDiagSlaveInfo.stState.bLinkError);
            fbJson.AddKey('Missing link');
            fbJson.AddBool(rDiagSlaveInfo.stState.bMissingLink);
            fbJson.AddKey('Unexpected link');
            fbJson.AddBool(rDiagSlaveInfo.stState.bUnexpectedLink);
            fbJson.AddKey('Port - A');
            fbJson.AddBool(rDiagSlaveInfo.stState.bPortA);
            fbJson.AddKey('Port - B');
            fbJson.AddBool(rDiagSlaveInfo.stState.bPortB);
            fbJson.AddKey('Port - C');
            fbJson.AddBool(rDiagSlaveInfo.stState.bPortC);
            fbJson.AddKey('Port - D');
            fbJson.AddBool(rDiagSlaveInfo.stState.bPortD);
    
        fbJson.EndObject();
    
    fbJson.EndObject();
    
fbJson.EndObject();

fbJson.CopyDocument(fbLogger.sJson, SIZEOF(fbLogger.sJson));
fbJson.ResetDocument();
END_ACTION

ACTION M_CheckMasterDevState:
(* check master errors based on devstate *)
bMasterDevStateError 				:= nMasterDevState <> 0;
stMasterDevState.bLinkError 		:= ((nMasterDevState AND 16#000F) = 1) OR ((nMasterDevState AND 16#000F) = 4);
stMasterDevState.bResetRequired 	:= ((nMasterDevState AND 16#000F) = 2) OR ((nMasterDevState AND 16#FFF0) = 16#10);
stMasterDevState.bMissFrmRedMode 	:= (nMasterDevState AND 16#000F) = 8;
stMasterDevState.bWatchdogTriggerd 	:= (nMasterDevState AND 16#20) = 16#20;
stMasterDevState.bDriverNotFound 	:= (nMasterDevState AND 16#40) = 16#40;
stMasterDevState.bResetActive 		:= (nMasterDevState AND 16#80) = 16#80;
stMasterDevState.bAtLeastOneNotInOp := ((nMasterDevState AND 16#100) = 16#100) OR ((nMasterDevState AND 16#200) = 16#200) OR
										((nMasterDevState AND 16#400) = 16#400) OR ((nMasterDevState AND 16#800) = 16#800);
stMasterDevState.bDcNotInSync 		:= (nMasterDevState AND 16#1000) = 16#1000;
nMasterDevStatePrev 				:= nMasterDevState;
END_ACTION

ACTION M_GetScannedSlaveName:

rSlaveInfoScanned REF= arrSlaveInfoScanned[aiDiagIndex[iIdx]];
rScannedSlaveInfo REF= arrScannedSlaveInfo[aiDiagIndex[iIdx]];

fbGetSlaveName(
	NETID		:= sIPCNetId,
	DEVICEID	:= nMasterDevID,
	BOXADDR		:= rScannedSlaveInfo.nAddr,
	START		:= TRUE,
	TMOUT		:= tTimeout,
	BOXNAME		=> strName
);

IF NOT fbGetSlaveName.BUSY THEN
	fbGetSlaveName(START:= FALSE);

	(* add scanned info *)
	rSlaveInfoScanned.nIndex 	:= iDiagIndex + 1;
	IF rScannedSlaveInfo.nAddr <> 0 THEN
		IF NOT fbGetSlaveName.ERR THEN
			rSlaveInfoScanned.sName := strName;
		END_IF
	ELSE
		rSlaveInfoScanned.sType		:= '';
	END_IF

	IF (iDiagIndex < nScannedSlaves) THEN
		rSlaveInfoScanned.sType		:= F_ConvProductCodeToString(rScannedSlaveInfo.stSlaveIdentity);
	ELSE
		rSlaveInfoScanned.sType		:= '';
	END_IF

	rSlaveInfoScanned.nECAddr	:= rScannedSlaveInfo.nAddr;

	IF rSlaveInfoScanned.sName <> rSlaveInfo.sName THEN
		rSlaveInfoScanned.bDifferentName := TRUE;
	ELSE
		rSlaveInfoScanned.bDifferentName := FALSE;
	END_IF

	IF rSlaveInfoScanned.nECAddr <> rSlaveInfo.nECAddr THEN
		rSlaveInfoScanned.bDifferentAddr := TRUE;
	ELSE
		rSlaveInfoScanned.bDifferentAddr := FALSE;
	END_IF

	IF rSlaveInfoScanned.sType <> rSlaveInfo.sType THEN
		rSlaveInfoScanned.bDifferentType := TRUE;
	ELSE
		rSlaveInfoScanned.bDifferentType := FALSE;
	END_IF

	IF iIdx < ESC_MAX_PORTS THEN
		iIdx := iIdx + 1;
		iState := E_EcatDiagState.GetSlaveIdentity; // loop back
	ELSE
		iIdx := 0;
		iState := E_EcatDiagState.LogDiagnostics;

		FOR I := 0 TO ESC_MAX_PORTS DO
			IF aiDiagPort[I] <> 0 THEN
				arrDiagSlaveInfo[I] := arrSlaveInfo[aiDiagIndex[I]];
				arrDiagSlaveInfoScanned[I] := arrSlaveInfoScanned[aiDiagIndex[I]];
			ELSE
				MEMSET(ADR(arrDiagSlaveInfo[I]), 0, SIZEOF(arrDiagSlaveInfo[I]));
				MEMSET(ADR(arrDiagSlaveInfoScanned[I]), 0, SIZEOF(arrDiagSlaveInfoScanned[I]));
			END_IF
		END_FOR
	END_IF
END_IF
END_ACTION

ACTION M_GetSlaveAdresses:
fbGetSlaveAddresses(
	sNetId		:= sMasterNetID,
	pAddrBuf	:= ADR(arrSlaveAddresses),
	cbBufLen	:= SIZEOF(arrSlaveAddresses),
	bExecute	:= TRUE,
	tTimeout	:= tTimeout,
	nSlaves		=> iNumOfSlavesRead
);

IF NOT fbGetSlaveAddresses.bBusy THEN
	fbGetSlaveAddresses(bExecute:= FALSE);
	IF NOT fbGetSlaveAddresses.bError THEN
		FOR I := 0 TO MIN(iNumOfSlavesRead, iSLAVEADDR_ARR_SIZE) DO
			arrSlaveInfo[I].nECAddr := arrSlaveAddresses[I];
		END_FOR
	END_IF
	iState := GetSlaveStates;
END_IF
END_ACTION

ACTION M_GetSlaveIdentity:

iDiagIndex := aiDiagIndex[iIdx];
iDiagPort := aiDiagPort[iIdx];

rSlaveInfo REF= arrSlaveInfo[iDiagIndex];

fbGetSlaveIdentity(
	sNetId		:= sMasterNetID,
	nSlaveAddr	:= rSlaveInfo.nECAddr,
	bExecute	:= TRUE,
	tTimeout	:= tTimeout,
	identity	=> stIdentity
);

IF NOT fbGetSlaveIdentity.bBusy THEN
	fbGetSlaveIdentity(bExecute:= FALSE);

	IF NOT fbGetSlaveIdentity.bError THEN
		IF aiDiagPort[iIdx] <> 0 THEN
			rSlaveInfo.nIndex	:= aiDiagIndex[iIdx] + 1;
			rSlaveInfo.sType 	:= F_ConvProductCodeToString(stSlaveIdentity := stIdentity);
		END_IF
	END_IF
	iState := E_EcatDiagState.GetSlaveName;
END_IF
END_ACTION

ACTION M_GetSlaveName:
fbGetSlaveName(
	NETID		:= sIPCNetId,
	DEVICEID	:= nMasterDevID,
	BOXADDR		:= rSlaveInfo.nECAddr,
	START		:= TRUE,
	TMOUT		:= tTimeout,
	BOXNAME		=> strName
);

IF NOT fbGetSlaveName.BUSY THEN
	fbGetSlaveName(START:= FALSE);

	IF NOT fbGetSlaveName.ERR THEN
		IF iDiagPort <> 0 THEN
			rSlaveInfo.sName 	:= strName;
		END_IF
	END_IF

	iState := E_EcatDiagState.GetScannedSlaveName;
END_IF
END_ACTION

ACTION M_GetSlaveStates:
fbGetAllSlaveStates(
	sNetId		:= sMasterNetID,
	pStateBuf	:= ADR(arrSlaveStates),
	cbBufLen	:= SIZEOF(arrSlaveStates),
	bExecute	:= TRUE,
	tTimeout	:= tTimeout,
	nSlaves		=> iNumOfSlavesRead
);

IF NOT fbGetAllSlaveStates.bBusy THEN
	fbGetAllSlaveStates(bExecute:= FALSE);

	IF NOT fbGetAllSlaveStates.bError THEN
		IF iNumOfSlavesRead = nSlaveCountCfg THEN
			FOR I := 0 TO ESC_MAX_PORTS DO
				aiDiagIndex[I] := 0;
			END_FOR

			(* split slave state and link state *)
			FOR I := 0 TO MIN(iNumOfSlavesRead, iSLAVEADDR_ARR_SIZE) DO
				(* slave state*)
				arrSlaveInfo[I].stState.eEcState 		:= arrSlaveStates[I].deviceState AND 16#0F;
				arrSlaveInfo[I].stState.bError 			:= arrSlaveStates[I].deviceState.4;
				arrSlaveInfo[I].stState.bInvalidVPRS 	:= arrSlaveStates[I].deviceState.5;
				(* link state *)
				arrSlaveInfo[I].stState.bNoCommToSlave 	:= arrSlaveStates[I].linkState.0;
				arrSlaveInfo[I].stState.bLinkError 		:= arrSlaveStates[I].linkState.1;
				arrSlaveInfo[I].stState.bMissingLink 	:= arrSlaveStates[I].linkState.2;
				arrSlaveInfo[I].stState.bUnexpectedLink := arrSlaveStates[I].linkState.3;
				arrSlaveInfo[I].stState.bPortA 			:= arrSlaveStates[I].linkState.4;
				arrSlaveInfo[I].stState.bPortB 			:= arrSlaveStates[I].linkState.5;
				arrSlaveInfo[I].stState.bPortC 			:= arrSlaveStates[I].linkState.6;
				arrSlaveInfo[I].stState.bPortD 			:= arrSlaveStates[I].linkState.7;
				(* DiagData *)
				arrSlaveInfo[I].bDiagData	:= ((arrSlaveStates[I].deviceState AND 16#F0) <> 0) OR
					(((arrSlaveStates[I].deviceState AND 16#0F) > 0) AND ((arrSlaveStates[I].deviceState AND 16#0F) < 8)) OR
					(arrSlaveStates[I].linkState <> 0);

				IF arrSlaveInfo[I].bDiagData THEN
					IF (I=0) THEN
						aiDiagIndex[0] := 0;
					ELSE
						IF (aiDiagIndex[0] = 0) AND NOT arrSlaveInfo[0].bDiagData THEN
							aiDiagIndex[0] :=  UDINT_TO_UINT(I);
						END_IF
					END_IF
				END_IF
			END_FOR
		END_IF
	END_IF

	IF arrSlaveInfo[aiDiagIndex[0]].bDiagData THEN
		iState := E_EcatDiagState.GetTopoDataLen;
	ELSE
		FOR I := 0 TO ESC_MAX_PORTS DO
			MEMSET(ADR(arrDiagSlaveInfo[I]), 0, SIZEOF(arrDiagSlaveInfo[I]));
			MEMSET(ADR(arrDiagSlaveInfoScanned[I]), 0, SIZEOF(arrDiagSlaveInfoScanned[I]));
		END_FOR
		iState := E_EcatDiagState.Done;
	END_IF
END_IF
END_ACTION

ACTION M_GetTopoData:
fbGetTopologyData(
	NETID	:= sMasterNetID,
	PORT	:= 16#FFFF,
	IDXGRP	:= 16#22,
	IDXOFFS	:= 0,
	LEN		:= iTopologyData*SIZEOF(arrTopologyData[0]),
	DESTADDR:= ADR(arrTopologyData),
	READ	:= TRUE,
	TMOUT	:= tTimeout,
);

IF NOT fbGetTopologyData.BUSY THEN
	fbGetTopologyData(READ := FALSE);

	IF NOT fbGetTopologyData.ERR THEN
		aiDiagPort[0] := arrTopologyData[aiDiagIndex[0]].iOwnPhysicalAddr;
		aiDiagPort[1] := arrTopologyData[aiDiagIndex[0]].stPhysicalAddr.portB;
		aiDiagPort[2] := arrTopologyData[aiDiagIndex[0]].stPhysicalAddr.portC;
		aiDiagPort[ESC_MAX_PORTS] := arrTopologyData[aiDiagIndex[0]].stPhysicalAddr.portD;

		(* clear diag index  *)
		aiDiagIndex[1] := 0;
		aiDiagIndex[2] := 0;
		aiDiagIndex[ESC_MAX_PORTS] := 0;
        
        (* find slaves on PortB-D of first slave with diag *)
        FOR P := 0 TO ESC_MAX_PORTS DO
            IF aiDiagPort[P] <> 0 THEN
			FOR I := 0 TO MIN(iTopologyData-1,iSLAVEADDR_ARR_SIZE) DO
				IF arrTopologyData[I].iOwnPhysicalAddr = aiDiagPort[P] THEN
					aiDiagIndex[P] := UDINT_TO_UINT(I);
					EXIT;
				END_IF
			END_FOR
		END_IF
		END_FOR
    END_IF

	iIdx := 0;
	iState := E_EcatDiagState.ScanSlaves;
END_IF
END_ACTION

ACTION M_GetTopoDataLen:
fbGetTopologyData(
	NETID	:= sMasterNetID,
	PORT	:= 16#FFFF,
	IDXGRP	:= EC_ADS_IGRP_MASTER_COUNT_SLAVE,
	IDXOFFS	:= EC_ADS_IOFFS_MASTER_COUNT_SLAVE,
	LEN		:= SIZEOF(iTopologyData),
	DESTADDR:= ADR(iTopologyData),
	READ	:= TRUE,
	TMOUT	:= tTimeout,
);

IF NOT fbGetTopologyData.BUSY THEN
	fbGetTopologyData(READ := FALSE);

	iState := E_EcatDiagState.GetTopoData;
END_IF
END_ACTION

ACTION M_ScanSlaves:
fbEcGetScannedSlaves(
	bExecute				:= TRUE,
	sNetId					:= sMasterNetID,
	pArrEcScannedSlaveInfo	:= ADR(arrScannedSlaveInfo),
	cbBufLen				:= SIZEOF(arrScannedSlaveInfo),
	tTimeout				:= tTimeout
);

IF NOT fbEcGetScannedSlaves.bBusy THEN
	fbEcGetScannedSlaves(bExecute := FALSE);
	
	IF fbEcGetScannedSlaves.bError THEN
		nScannedSlaves := 0;
	ELSE
		nScannedSlaves := fbEcGetScannedSlaves.nSlaves;
	END_IF
    
    iState := E_EcatDiagState.GetSlaveIdentity;
    
END_IF
END_ACTION

END_FUNCTION_BLOCK

// EtherCatDiagnostic/FB_EtherCATDiagnosticWrapper
FUNCTION_BLOCK FB_EtherCATDiagnosticWrapper
VAR_INPUT
	nEcMasterSlaveCount  	AT%I*: UINT;				// link to SlaveCount of EtherCAT Master (Inputs) {attribute 'TcLinkTo' := 'TIID^Device 1 (EtherCAT)^Inputs^SlaveCount'}
	nEcMasterDevState 		AT%I*: UINT;				// link to DevState of EtherCAT Master (Inputs) {attribute 'TcLinkTo' := 'TIID^Device 1 (EtherCAT)^Inputs^DevState'}
	nEcMasterDeviceId 		AT%I*: UINT;				// link to DevID of EtherCAT Master (InfoData)  {attribute 'TcLinkTo' := 'TIID^Device 1 (EtherCAT)^InfoData^DevId'}
	arrEcMasterNetId  		AT%I*: T_AmsNetIdArr;	// link to NetID of EtherCAT Master (InfoData)	{attribute 'TcLinkTo' := 'TIID^Device 1 (EtherCAT)^InfoData^AmsNetId'}
	nEcMasterSlaveCountCfg  AT%I*: UINT;				// link to CfgSlaveCount of EtherCAT Master (InfoData) {attribute 'TcLinkTo' := 'TIID^Device 1 (EtherCAT)^InfoData^CfgSlaveCount'}
	
	(* ******************* EtherCAT Frame ***************************** *)
	wFrmXWcState 			AT%I*: WORD; 			// link to task related ethercat frame state (Frm1WcState) {attribute 'TcLinkTo' := 'TIID^Device 1 (EtherCAT)^Inputs^Frm1WcState'} 
END_VAR
VAR_OUTPUT
    bAllFrameWcStatesOK		: BOOL;				// all frames are OK
    bEtherCATOK				: BOOL;				// no problem on EtherCAT
	bFrameWcStateError		: BOOL;				// at least one fram with error
	bSlaveCountError		: BOOL;				// EtherCAT slave count mismatch (# of cfg slaves <> # of found slaves)
	bMasterDevStateError	: BOOL;				// EtherCAT master device state signals error
	stMasterDevState		: ST_EcMasterDevState; // device state split to a structure
	bBusy					: BOOL;				// diagnostic FB is busy
	bError					: BOOL;				// diagnostic FB has an error
	iErrorID				: UDINT;			// error ID of diagnostic FB
END_VAR
VAR_IN_OUT
	arrSlaveInfo			: ARRAY [0..iSLAVEADDR_ARR_SIZE] OF ST_SlaveStateInfo; 
END_VAR
VAR
    sEcMasterNetId  		: T_AmsNetId := '';
    (* ******************* EtherCAT Frame ***************************** *)
	fbEtherCATFrameDiag		: FB_EtherCATFrameDiag; 	// frame diagnostic

	wReqZeroMask			: WORD := 16#FFFF; 			// clear bit to ignore datagram error of Frm1WcState
	bFrameWcStateOK			: BOOL;						// this frame is OK 

    (* ******************* EtherCAT Diag ***************************** *)
    fbEtherCATDiag			: FB_EtherCATDiag;			// deep EtherCAT diagnostic
	fbEtherCATSlaveInfo		: FB_EtherCATSlaveInfo;		// slave info collector

	(* general variables *)
	arrDiagSlaveInfo 			: ARRAY [0..ESC_MAX_PORTS] OF ST_SlaveStateInfo;		// read in info of configured EtherCAT slaves 
	arrDiagSlaveInfoScanned		: ARRAY [0..ESC_MAX_PORTS] OF ST_SlaveStateInfoScanned; // read in info of scanned EtherCAT slaves  
END_VAR


(*************************************** Frame Diag *********************************************)
fbEtherCATFrameDiag(
	wFrmXWcState 	:= wFrmXWcState,
	wReqZeroMask 	:= wReqZeroMask,
	bFrameWcStateOK	=> bFrameWcStateOK
);
bAllFrameWcStatesOK := bFrameWcStateOK;

(*************************************** EtherCAT Diag *********************************************)
(* generate Net Id *)
sEcMasterNetId := F_CreateAmsNetId(nIds := arrEcMasterNetId);
fbEtherCATDiag(
	sIPCNetID			:= '',
	sMasterNetID		:= sEcMasterNetId,
	nMasterDevID		:= nEcMasterDeviceId,
	nSlaveCount			:= nEcMasterSlaveCount,
	nSlaveCountCfg		:= nEcMasterSlaveCountCfg,
	nMasterDevState		:= nEcMasterDevState,
	bAllFrameWcStatesOK	:= bAllFrameWcStatesOK,
	tTimeout			:= T#5s,
	arrDiagSlaveInfo	:= arrDiagSlaveInfo,
	arrDiagSlaveInfoScanned	:= arrDiagSlaveInfoScanned,
	bEtherCATOK			=> bEtherCATOK,
	bFrameWcStateError	=> bFrameWcStateError,
	bSlaveCountError	=> bSlaveCountError,
	bMasterDevStateError=> bMasterDevStateError,
	stMasterDevState	=> stMasterDevState,
	bBusy				=> bBusy,
	bError				=> bError,
	iErrorID			=> iErrorID
);
fbEtherCATSlaveInfo(
	sIPCNetID			:= '',
	sMasterNetID		:= sEcMasterNetId,
	nMasterDevID		:= nEcMasterDeviceId,
	nSlaveCount			:= nEcMasterSlaveCount,
	nSlaveCountCfg		:= nEcMasterSlaveCountCfg,
	nMasterDevState		:= nEcMasterDevState,
	bAllFrameWcStatesOK	:= bAllFrameWcStatesOK,
	tTimeout			:= T#5s,
	arrSlaveInfo		:= arrSlaveInfo
);

END_FUNCTION_BLOCK

// EtherCatDiagnostic/FB_EtherCATFrameDiag
FUNCTION_BLOCK FB_EtherCATFrameDiag
VAR_INPUT
	wFrmXWcState 		: WORD;				// FrmXWcState
	wReqZeroMask 		: WORD := 16#FFFF;	// mask, bit TRUE: require wFrmXWcState.bit = FALSE, bit FALSE: ignore wFrmXWcState.bit *)
END_VAR
VAR_OUTPUT
	bFrameWcStateOK		: BOOL;				// result of fram state check
END_VAR
VAR
END_VAR

(* mask out ignored error bits and compare result against 0 *)
bFrameWcStateOK := ((wFrmXWcState AND wReqZeroMask) = 0);

END_FUNCTION_BLOCK

// EtherCatDiagnostic/FB_EtherCATSlaveInfo
FUNCTION_BLOCK FB_EtherCATSlaveInfo
VAR_INPUT
	sIPCNetID					: T_AmsNetId; 	// AmsNetId of the IPC 
	sMasterNetID				: T_AmsNetId; 	// AmsNetId of the EtherCAT master device 
	nMasterDevID				: UINT;			// Device ID of EtherCAT master
	nSlaveCount 				: UINT;			// current slave count
	nSlaveCountCfg 				: UINT;			// configured slave count
	nMasterDevState				: WORD;			// device state of EtherCAT Master
	bAllFrameWcStatesOK			: BOOL;			// all FrameWcState OK?
	tTimeout					: TIME := T#5S; // ads timeout
END_VAR
VAR_OUTPUT
	bEtherCATOK					: BOOL;			// no problem on EtherCAT
	bFrameWcStateError			: BOOL;			// error in at least one frame
	bSlaveCountError			: BOOL;			// EtherCAT slave count mismatch (# of cfg slaves <> # of found slaves)
	bMasterDevStateError		: BOOL;			// error in master device state
	stMasterDevState			: ST_EcMasterDevState; // splitted master device state
	bBusy						: BOOL;			// FB busy
	bError						: BOOL;			// FB with error
	iErrorID					: UDINT;		// FB error ID
END_VAR

VAR_IN_OUT
	arrSlaveInfo 			: ARRAY [0..iSLAVEADDR_ARR_SIZE] OF ST_SlaveStateInfo;		// read in info from configured slaves
END_VAR
VAR
	sMasterOpState				: STRING(255);
	sSlaveOpState				: STRING(255);
	iState						: E_EcatDiagState;
	nMasterDevStatePrev			: WORD;
	bSlaveCountErrorPrev		: BOOL;
	bAllFrameWcStatesOKPrev		: BOOL;
	bDiagReq					: BOOL := TRUE;
	I							: UDINT;
    P							: UDINT;
    rSlaveInfo  				: REFERENCE TO ST_SlaveStateInfo;

	(* -- Get Slave Addresses *)
	fbGetSlaveAddresses 		: FB_EcGetAllSlaveAddr;
	arrSlaveAddresses 			: ARRAY[0..iSLAVEADDR_ARR_SIZE] OF UINT;
	iNumOfSlavesRead			: UINT;

	(* -- Get Slave States *)
	fbGetAllSlaveStates			: FB_EcGetAllSlaveStates;
	arrSlaveStates 				: ARRAY[0..iSLAVEADDR_ARR_SIZE] OF ST_EcSlaveState;

	(* -- Get Topology Data *)
	iTopologyData				: UDINT;
	fbGetTopologyData			: ADSREAD;
	arrTopologyData				: ARRAY[0..iSLAVEADDR_ARR_SIZE] OF ST_TopologyData;

	(* -- Check Topology *)
	aiDiagIndex					: ARRAY [0..ESC_MAX_PORTS] OF UINT;
    iDiagIndex 					: UINT;    
	aiDiagPort					: ARRAY [0..ESC_MAX_PORTS] OF UINT;
    iDiagPort 					: UINT;
	iIdx						: DINT;

	(* -- Scan Slaves *)
	fbEcGetScannedSlaves		: FB_EcGetScannedSlaves;
	arrScannedSlaveInfo			: ARRAY [0..iSLAVEADDR_ARR_SIZE] OF ST_EcSlaveScannedData; // what...
    rScannedSlaveInfo   		: REFERENCE TO ST_EcSlaveScannedData;
	nScannedSlaves				: UINT;

	(* -- Get Slave Identities *)
	fbGetSlaveIdentity			: FB_EcGetSlaveIdentity;
	stIdentity 					: ST_EcSlaveIdentity;

	(* -- Get Slave Names *)
	fbGetSlaveName 				: IOF_GetBoxNameByAddr;
    arrSlaveInfoScanned			: ARRAY [0..iSLAVEADDR_ARR_SIZE] OF ST_SlaveStateInfoScanned; // the F
    rSlaveInfoScanned   		: REFERENCE TO ST_SlaveStateInfoScanned;
	strName						: STRING;

    // Logging components
    rDiagSlaveInfo 				: REFERENCE TO ST_SlaveStateInfo;
    tEtherCATOK 				: F_TRIG;
    tFrameWcStateError 			: R_TRIG;
    tMasterError 				: R_TRIG;
	tpQuerryTrigger				: TP;
END_VAR

tpQuerryTrigger(IN:=tpQuerryTrigger.Q, PT:=T#500MS);

(* acyclic diag *)
CASE iState OF
E_EcatDiagState.Idle: (* IDLE *)
	IF NOT tpQuerryTrigger.Q THEN
		bBusy := TRUE;
		iState:=E_EcatDiagState.GetSlaveAddresses;
	END_IF
E_EcatDiagState.GetSlaveAddresses: (* get adresses *)
	M_GetSlaveAdresses();

E_EcatDiagState.GetSlaveStates: (* get states *)
	M_GetSlaveStates();

E_EcatDiagState.GetTopoDataLen:	(* get topology data length *)
	M_GetTopoDataLen();

E_EcatDiagState.GetTopoData:	(* get topology data *)
	M_GetTopoData();

E_EcatDiagState.ScanSlaves:	(* scan slaves *)
	M_ScanSlaves();

E_EcatDiagState.GetSlaveIdentity:	(* get identity *)
	M_GetSlaveIdentity();

E_EcatDiagState.GetSlaveName:	(* get name *)
	M_GetSlaveName();

E_EcatDiagState.GetScannedSlaveName:	(* get scanned name *)
	M_GetScannedSlaveName();  
    
E_EcatDiagState.Done:	(* DONE *)
	bBusy := FALSE;
	iState := 0;
END_CASE

ACTION M_GetScannedSlaveName:

rSlaveInfoScanned REF= arrSlaveInfoScanned[iIdx];
rScannedSlaveInfo REF= arrScannedSlaveInfo[iIdx];

fbGetSlaveName(
	NETID		:= sIPCNetId,
	DEVICEID	:= nMasterDevID,
	BOXADDR		:= rScannedSlaveInfo.nAddr,
	START		:= TRUE,
	TMOUT		:= tTimeout,
	BOXNAME		=> strName
);

IF NOT fbGetSlaveName.BUSY THEN
	fbGetSlaveName(START:= FALSE);

	(* add scanned info *)
	rSlaveInfoScanned.nIndex 	:= iDiagIndex + 1;
	IF rScannedSlaveInfo.nAddr <> 0 THEN
		IF NOT fbGetSlaveName.ERR THEN
			rSlaveInfoScanned.sName := strName;
		END_IF
	ELSE
		rSlaveInfoScanned.sType		:= '';
	END_IF

	IF (iIdx < nScannedSlaves) THEN
		rSlaveInfoScanned.sType		:= F_ConvProductCodeToString(rScannedSlaveInfo.stSlaveIdentity);
	ELSE
		rSlaveInfoScanned.sType		:= '';
	END_IF

	rSlaveInfoScanned.nECAddr	:= rScannedSlaveInfo.nAddr;

	IF rSlaveInfoScanned.sName <> rSlaveInfo.sName THEN
		rSlaveInfoScanned.bDifferentName := TRUE;
	ELSE
		rSlaveInfoScanned.bDifferentName := FALSE;
	END_IF

	IF rSlaveInfoScanned.nECAddr <> rSlaveInfo.nECAddr THEN
		rSlaveInfoScanned.bDifferentAddr := TRUE;
	ELSE
		rSlaveInfoScanned.bDifferentAddr := FALSE;
	END_IF

	IF rSlaveInfoScanned.sType <> rSlaveInfo.sType THEN
		rSlaveInfoScanned.bDifferentType := TRUE;
	ELSE
		rSlaveInfoScanned.bDifferentType := FALSE;
	END_IF

	IF iIdx < MIN(iSLAVEADDR_ARR_SIZE,iNumOfSlavesRead) THEN
		iIdx := iIdx + 1;
		iState := E_EcatDiagState.GetSlaveIdentity; // loop back
	ELSE
		iIdx := 0;
		iState := E_EcatDiagState.Done;
	END_IF
END_IF
END_ACTION

ACTION M_GetSlaveAdresses:
fbGetSlaveAddresses(
	sNetId		:= sMasterNetID,
	pAddrBuf	:= ADR(arrSlaveAddresses),
	cbBufLen	:= SIZEOF(arrSlaveAddresses),
	bExecute	:= TRUE,
	tTimeout	:= tTimeout,
	nSlaves		=> iNumOfSlavesRead
);

IF NOT fbGetSlaveAddresses.bBusy THEN
	fbGetSlaveAddresses(bExecute:= FALSE);
	IF NOT fbGetSlaveAddresses.bError THEN
		FOR I := 0 TO MIN(iNumOfSlavesRead, iSLAVEADDR_ARR_SIZE) DO
			arrSlaveInfo[I].nECAddr := arrSlaveAddresses[I];
		END_FOR
	END_IF
	iState := GetSlaveStates;
END_IF
END_ACTION

ACTION M_GetSlaveIdentity:
rSlaveInfo REF= arrSlaveInfo[iIdx];

fbGetSlaveIdentity(
	sNetId		:= sMasterNetID,
	nSlaveAddr	:= rSlaveInfo.nECAddr,
	bExecute	:= TRUE,
	tTimeout	:= tTimeout,
	identity	=> stIdentity
);

IF NOT fbGetSlaveIdentity.bBusy THEN
	fbGetSlaveIdentity(bExecute:= FALSE);

	IF NOT fbGetSlaveIdentity.bError THEN
		rSlaveInfo.nIndex	:= iIdx;
		rSlaveInfo.sType 	:= F_ConvProductCodeToString(stSlaveIdentity := stIdentity);
	END_IF
	iState := E_EcatDiagState.GetSlaveName;
END_IF
END_ACTION

ACTION M_GetSlaveName:
fbGetSlaveName(
	NETID		:= sIPCNetId,
	DEVICEID	:= nMasterDevID,
	BOXADDR		:= rSlaveInfo.nECAddr,
	START		:= TRUE,
	TMOUT		:= tTimeout,
	BOXNAME		=> strName
);

IF NOT fbGetSlaveName.BUSY THEN
	fbGetSlaveName(START:= FALSE);

	IF NOT fbGetSlaveName.ERR THEN
		rSlaveInfo.sName 	:= strName;
	END_IF

	iState := E_EcatDiagState.GetScannedSlaveName;
END_IF
END_ACTION

ACTION M_GetSlaveStates:
fbGetAllSlaveStates(
	sNetId		:= sMasterNetID,
	pStateBuf	:= ADR(arrSlaveStates),
	cbBufLen	:= SIZEOF(arrSlaveStates),
	bExecute	:= TRUE,
	tTimeout	:= tTimeout,
	nSlaves		=> iNumOfSlavesRead
);

IF NOT fbGetAllSlaveStates.bBusy THEN
	fbGetAllSlaveStates(bExecute:= FALSE);

	IF NOT fbGetAllSlaveStates.bError THEN
		IF iNumOfSlavesRead = nSlaveCountCfg THEN
			FOR I := 0 TO ESC_MAX_PORTS DO
				aiDiagIndex[I] := 0;
			END_FOR

			(* split slave state and link state *)
			FOR I := 0 TO MIN(iNumOfSlavesRead, iSLAVEADDR_ARR_SIZE) DO
				(* slave state*)
				arrSlaveInfo[I].stState.eEcState 		:= arrSlaveStates[I].deviceState AND 16#0F;
				arrSlaveInfo[I].stState.bError 			:= arrSlaveStates[I].deviceState.4;
				arrSlaveInfo[I].stState.bInvalidVPRS 	:= arrSlaveStates[I].deviceState.5;
				(* link state *)
				arrSlaveInfo[I].stState.bNoCommToSlave 	:= arrSlaveStates[I].linkState.0;
				arrSlaveInfo[I].stState.bLinkError 		:= arrSlaveStates[I].linkState.1;
				arrSlaveInfo[I].stState.bMissingLink 	:= arrSlaveStates[I].linkState.2;
				arrSlaveInfo[I].stState.bUnexpectedLink := arrSlaveStates[I].linkState.3;
				arrSlaveInfo[I].stState.bPortA 			:= arrSlaveStates[I].linkState.4;
				arrSlaveInfo[I].stState.bPortB 			:= arrSlaveStates[I].linkState.5;
				arrSlaveInfo[I].stState.bPortC 			:= arrSlaveStates[I].linkState.6;
				arrSlaveInfo[I].stState.bPortD 			:= arrSlaveStates[I].linkState.7;
			END_FOR
		END_IF
	END_IF
	iState := E_EcatDiagState.GetTopoDataLen;
END_IF
END_ACTION

ACTION M_GetTopoData:
fbGetTopologyData(
	NETID	:= sMasterNetID,
	PORT	:= 16#FFFF,
	IDXGRP	:= 16#22,
	IDXOFFS	:= 0,
	LEN		:= iTopologyData*SIZEOF(arrTopologyData[0]),
	DESTADDR:= ADR(arrTopologyData),
	READ	:= TRUE,
	TMOUT	:= tTimeout,
);

IF NOT fbGetTopologyData.BUSY THEN
	fbGetTopologyData(READ := FALSE);

	IF NOT fbGetTopologyData.ERR THEN
		aiDiagPort[0] := arrTopologyData[aiDiagIndex[0]].iOwnPhysicalAddr;
		aiDiagPort[1] := arrTopologyData[aiDiagIndex[0]].stPhysicalAddr.portB;
		aiDiagPort[2] := arrTopologyData[aiDiagIndex[0]].stPhysicalAddr.portC;
		aiDiagPort[ESC_MAX_PORTS] := arrTopologyData[aiDiagIndex[0]].stPhysicalAddr.portD;

		(* clear diag index  *)
		aiDiagIndex[1] := 0;
		aiDiagIndex[2] := 0;
		aiDiagIndex[ESC_MAX_PORTS] := 0;
        
        (* find slaves on PortB-D of first slave with diag *)
        FOR P := 0 TO ESC_MAX_PORTS DO
            IF aiDiagPort[P] <> 0 THEN
			FOR I := 0 TO MIN(iTopologyData-1,iSLAVEADDR_ARR_SIZE) DO
				IF arrTopologyData[I].iOwnPhysicalAddr = aiDiagPort[P] THEN
					aiDiagIndex[P] := UDINT_TO_UINT(I);
					EXIT;
				END_IF
			END_FOR
		END_IF
		END_FOR
    END_IF

	iIdx := 0;
	iState := E_EcatDiagState.ScanSlaves;
END_IF
END_ACTION

ACTION M_GetTopoDataLen:
fbGetTopologyData(
	NETID	:= sMasterNetID,
	PORT	:= 16#FFFF,
	IDXGRP	:= EC_ADS_IGRP_MASTER_COUNT_SLAVE,
	IDXOFFS	:= EC_ADS_IOFFS_MASTER_COUNT_SLAVE,
	LEN		:= SIZEOF(iTopologyData),
	DESTADDR:= ADR(iTopologyData),
	READ	:= TRUE,
	TMOUT	:= tTimeout,
);

IF NOT fbGetTopologyData.BUSY THEN
	fbGetTopologyData(READ := FALSE);

	iState := E_EcatDiagState.GetTopoData;
END_IF
END_ACTION

ACTION M_ScanSlaves:
fbEcGetScannedSlaves(
	bExecute				:= TRUE,
	sNetId					:= sMasterNetID,
	pArrEcScannedSlaveInfo	:= ADR(arrScannedSlaveInfo),
	cbBufLen				:= SIZEOF(arrScannedSlaveInfo),
	tTimeout				:= tTimeout
);

IF NOT fbEcGetScannedSlaves.bBusy THEN
	fbEcGetScannedSlaves(bExecute := FALSE);
	
	IF fbEcGetScannedSlaves.bError THEN
		nScannedSlaves := 0;
	ELSE
		nScannedSlaves := fbEcGetScannedSlaves.nSlaves;
	END_IF
    
    iState := E_EcatDiagState.GetSlaveIdentity;
    
END_IF
END_ACTION

END_FUNCTION_BLOCK

// EventLogger/FB_EventHandler
FUNCTION_BLOCK FB_EventHandler
VAR_INPUT
	bClearAll:				BOOL;
END_VAR
VAR_OUTPUT
	bAlarmActive:			BOOL;	
	sEventText:				STRING(255);
	sEventSource:			STRING(255);
	sEventJson:				STRING(7000);
END_VAR
VAR
	rtClear:				R_TRIG;
	FB_TcEventLogger:		FB_TcEventLogger;
END_VAR

rtClear(CLK:=bClearAll);

bAlarmActive:=EVENT_GVL.G_bAlarmActive;
sEventText:=EVENT_GVL.G_sAlarmMessage;
sEventSource:=EVENT_GVL.G_sAlarmSource;
sEventJson:=EVENT_GVL.G_sAlarmJson;

IF rtClear.Q THEN
	FB_TcEventLogger.ConfirmAllAlarms(0);
	FB_TcEventLogger.ClearAllAlarms(0, TRUE);
	EVENT_GVL.G_sAlarmJson:='';
	EVENT_GVL.G_sAlarmSource:='';
	EVENT_GVL.G_sAlarmMessage:='';
	EVENT_GVL.G_bAlarmActive:=FALSE;
END_IF

END_FUNCTION_BLOCK

// RecipeManager/FB_RecipeManager
{attribute 'reflection'}
FUNCTION_BLOCK FB_RecipeManager
VAR_INPUT
	sDef:				STRING(MAX_STRING_LENGTH):='DefaultsDef';
	sExt:				STRING(MAX_STRING_LENGTH):='tcdata';
	sFolderPath:		STRING(MAX_STRING_LENGTH):='C:\TwinCAT\Tc_Data';
	sKey:				STRING(MAX_STRING_LENGTH):='Data';
	pData:				PVOID;
	nData:				UDINT;
	RESET:				BOOL;
END_VAR
VAR_OUTPUT
	READY:				BOOL;
	BUSY:				BOOL;
	DONE:				BOOL;
	
	ERROR:				BOOL;
	ERROR_ID:			UDINT;
	
	TIME_STAMP:			STRING(MAX_STRING_LENGTH);
	RECIPE_LIST:		ARRAY[1..200] OF STRING;
	RECIPE_CNT:			UDINT;
END_VAR
VAR
	FB_SYSTIME: 		FB_LocalSystemTime:= (bEnable:= TRUE, dwCycle:= 1);
	WRITE_FILE:			FB_WriteTextFile;
	READ_FILE:			FB_ReadTextFile;
	RT_READ_FILE_ERROR:	R_TRIG;
	RT_WRITE_FILE_ERROR:R_TRIG;
	
	JSON_STRING:		STRING(MAX_JSON_LENGTH);
	JSON_LENGTH:		UDINT;
	
	STATE:				INT;
	INIT:				BOOL:=TRUE;
	EXECUTE:			BOOL;
	
	FILE_PATH:			STRING(MAX_STRING_LENGTH);
	FILE_NAME:			STRING(MAX_STRING_LENGTH);
	RECIPE_NAME:		STRING(MAX_STRING_LENGTH):='DefaultName';
	RECIPE_VALID:		BOOL;
	FB_CreateDir: 			FB_CreateDir;
	FB_FIND_FILE: 			FB_EnumFindFileEntry:= (sNetID:= '', tTimeout:= DEFAULT_ADS_TIMEOUT);
	ENUM_FIND_FILE:			STRING(MAX_STRING_LENGTH);
	ENUM_FIND_RECIPENAME:	STRING;
	ENUM_INDEX:				UDINT:=1;
	ENUMERATE: 				BOOL;
	ENUM_STATE: 			INT;
	
	eSubSystem: 			E_SubSystem:= E_SubSystem.LOGIC;
	FB_LOGGER:				FB_EventLogger:= (eSubsystem:= eSubsystem, sJson:='{}');
END_VAR

CREATE_PATH();
FB_FIND_FILE(sPathName:= CONCAT(sFolderPath, CONCAT('\', CONCAT('*', CONCAT('.', CONCAT(sDef, CONCAT('.', sExt)))))));
FB_SYSTIME();
READY:= STATE=0;
BUSY:= STATE<>0;

RT_READ_FILE_ERROR(CLK:=READ_FILE.ERROR);
IF RT_READ_FILE_ERROR.Q THEN
	ERROR_ID:=READ_FILE.ERROR_ID;
END_IF

RT_WRITE_FILE_ERROR(CLK:=WRITE_FILE.ERROR);
IF RT_WRITE_FILE_ERROR.Q THEN
	ERROR_ID:=WRITE_FILE.ERROR_ID;
END_IF

IF RESET THEN
	STATE:=0;
	ERROR_ID:=0;
	DONE:=FALSE;
END_IF

IF INIT THEN
	INIT := FALSE;
    FB_CreateDir( bExecute := FALSE );
    FB_CreateDir(sNetId:= '',
                sPathName:= sFolderPath,
                ePath:= PATH_GENERIC,
                bExecute:= TRUE,
                tTimeout:= DEFAULT_ADS_TIMEOUT);
ELSE
    FB_CreateDir(bExecute := FALSE);
END_IF

CASE STATE OF
	1100:
		CREATE_PATH();
		IF ANY_TO_JSON(pData,nData, sKey:=sKey, SYSTEMTIME_TO_STRING(FB_SYSTIME.systemTime), JSON_STRING, JSON_LENGTH) THEN
			STATE:=1200;
		END_IF
	1200:
		IF WRITE_FILE.Write(FILE_PATH) THEN
			STATE:=1300;
		END_IF
	2100:
		CREATE_PATH();
		//Refresh recipe lists
		IF ENUM_STATE=3 THEN
			ENUMERATE:=FALSE;
			STATE:=2200;
		END_IF
	2200:
		//Validate recipe
		IF ValidateRecipe(RECIPE_NAME, RECIPE_VALID) THEN
			IF RECIPE_VALID THEN
				STATE:=2300;
			ELSE
				FB_LOGGER(sMsg:=CONCAT(CONCAT('File not found. Invalid file name or file path. Error id: ', DWORD_TO_HEXSTR(ERROR_ID, 0, FALSE )),CONCAT(' Path: ', FILE_PATH)), eSevr:=TcEventSeverity.Error);
				ERROR_ID:=1804;
				STATE:=9999;
			END_IF
		END_IF
	2300:
		CREATE_PATH();
		IF READ_FILE.Read(FILE_PATH) THEN
			STATE:=2400;
		END_IF
	2400:
		IF JSON_TO_ANY(pData,nData, sKey:=sKey, TIME_STAMP, JSON_STRING) THEN
			EXECUTE:=FALSE;
			STATE:=2500;
		END_IF
	3100:
		ENUMERATE:=TRUE;
		STATE:=3200;
	3200:
		IF ENUM_STATE=3 THEN
			ENUMERATE:=FALSE;
			STATE:=3300;
		END_IF
	9999:
		//Error state pleaceholder
END_CASE

ERROR:=(ERROR_ID<>0);
ENUM_FILE_LIST_ACT();
FB_CALL_ACT();

ACTION ENUM_FILE_LIST_ACT:
CASE ENUM_STATE OF
	0:
		IF ENUMERATE THEN
			MEMSET(ADR(RECIPE_LIST), 0, SIZEOF(RECIPE_LIST));
			ENUM_INDEX:=1;
			FB_FIND_FILE.eCmd := eEnumCmd_First;
			ENUM_STATE := 1;
        END_IF
	1: 
        FB_FIND_FILE( bExecute := FALSE );
        FB_FIND_FILE( bExecute := TRUE );
        ENUM_STATE := 2;

	2:
		FB_FIND_FILE( bExecute := FALSE );
		IF NOT FB_FIND_FILE.bBusy THEN
			IF NOT FB_FIND_FILE.bError THEN
				IF NOT FB_FIND_FILE.bEOE THEN
					RECIPE_CNT:=ENUM_INDEX;
					ENUM_FIND_FILE:=FB_FIND_FILE.stFindFile.sFileName;					
					ENUM_FIND_RECIPENAME:=LEFT(FB_FIND_FILE.stFindFile.sFileName, (FIND(FB_FIND_FILE.stFindFile.sFileName, '.')-1));
					
					RECIPE_LIST[ENUM_INDEX]:=ENUM_FIND_RECIPENAME;
					FB_FIND_FILE.eCmd := eEnumCmd_Next;
					ENUM_INDEX:=ENUM_INDEX+1;
					ENUM_STATE:= 1;
				ELSE
					RECIPE_CNT:= ENUM_INDEX-1;
					ENUM_STATE := 3;
				END_IF
			ELSE
				ADSLOGSTR( ADSLOG_MSGTYPE_ERROR OR ADSLOG_MSGTYPE_LOG, 'FB_EnumFindFileEntry error:%s', DWORD_TO_HEXSTR( FB_FIND_FILE.nErrID, 0, FALSE ));
				ENUM_STATE := 3;
			END_IF
        END_IF
	3:
		IF NOT ENUMERATE THEN
			ENUM_STATE := 0;
		END_IF
END_CASE
END_ACTION

ACTION FB_CALL_ACT:
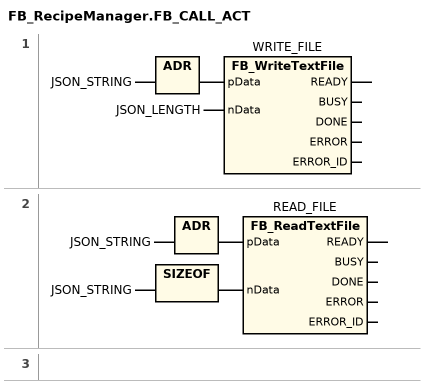
// NETWORK 1
WRITE_FILE(pData := ADR(JSON_STRING), nData := JSON_LENGTH); // FB_WriteTextFile

// NETWORK 2
READ_FILE(pData := ADR(JSON_STRING), nData := SIZEOF(JSON_STRING)); // FB_ReadTextFile

// NETWORK 3
END_ACTION

METHOD PRIVATE CREATE_PATH : BOOL
VAR_INPUT
END_VAR
FILE_NAME:=CONCAT(RECIPE_NAME, CONCAT('.', CONCAT(sDef, CONCAT('.', sExt))));
FILE_PATH:=CONCAT(sFolderPath, CONCAT('\', FILE_NAME));
END_METHOD

METHOD PUBLIC Load : BOOL
VAR_INPUT
	NAME:				STRING;
END_VAR
VAR
END_VAR
IF STATE=0 THEN
	DONE:=FALSE;
	RECIPE_VALID:=FALSE;
	RECIPE_NAME:=NAME;
	ENUMERATE:=TRUE;
	STATE:=2100;
END_IF

IF STATE=2500 THEN
	STATE:=0;
	DONE:=TRUE;
	Load:=TRUE;
	RETURN;
END_IF
END_METHOD

METHOD PUBLIC RefreshNameList : BOOL
VAR_INPUT
END_VAR
IF STATE=0 THEN
	DONE:=FALSE;
	STATE:=3100;
END_IF
IF STATE=3300 THEN
	DONE:=TRUE;
	STATE:=0;
	RefreshNameList:=TRUE;
	RETURN;
END_IF
END_METHOD

METHOD PUBLIC Save : BOOL
VAR_INPUT
	NAME:				STRING;
END_VAR
VAR
END_VAR
IF STATE=0 THEN
	DONE:=FALSE;
	RECIPE_NAME:=NAME;
	STATE:=1100;
END_IF
IF STATE=1300 THEN
	DONE:=TRUE;
	STATE:=0;
	Save:=TRUE;
	RETURN;
END_IF
END_METHOD

METHOD PUBLIC ValidateRecipe : BOOL
VAR_INPUT
	RECIPE_NAME:		REFERENCE TO STRING;
	IS_VLAID:			REFERENCE TO BOOL;
END_VAR
VAR
	CNT:				UDINT;
END_VAR
//Iterate trough the recipe name list, if find matching recipe return true else throw an error.
CNT:=1;
IS_VLAID:=FALSE;

FOR CNT:=1 TO RECIPE_CNT DO
    IF RECIPE_LIST[CNT] = RECIPE_NAME THEN
		IS_VLAID:=TRUE;
	END_IF
END_FOR;

ValidateRecipe:=TRUE;
END_METHOD

END_FUNCTION_BLOCK

// Tcp Barcode Reader/FB_BARCODE_READER
FUNCTION_BLOCK FB_BARCODE_READER
VAR_INPUT
	HOST:				T_IPV4ADDR := '';
	PORT:				UDINT;
	RESET:				BOOL;
END_VAR
VAR_OUTPUT
	BUSY:				BOOL;
	READY:				BOOL;
	DONE:				BOOL;
	
	ERROR:				BOOL;
	ERROR_ID:			UDINT;
	
	BARCODE:			STRING;
END_VAR
VAR
	FB_TCP_CLIENT:		FB_TCP_IP_CLIENT;
	STATE:				UDINT;
	TCP_BUFF:			STRING[DEFAULT_SDAT_LENGTH];
	STR_LON:			STRING[DEFAULT_SDAT_LENGTH]:='LON';
	STR_LOFF:			STRING[DEFAULT_SDAT_LENGTH]:='LOFF';
	SUB_SYS: 			E_SubSystem:= E_SubSystem.LOGIC;
	FB_LOGGER:			FB_EventLogger:= (eSubsystem:= SUB_SYS, sJson:='{}');
	RT_RESET:			R_TRIG;
END_VAR

RT_RESET(CLK:=RESET);

BUSY:= STATE <> 0;
READY:= STATE = 0;
ERROR:= ERROR_ID<>0;

IF ERROR_ID<>0 THEN
	STATE:=9999;
END_IF

IF RT_RESET.Q THEN
	MEMSET(ADR(TCP_BUFF),0,SIZEOF(TCP_BUFF));
	MEMSET(ADR(BARCODE),0,SIZEOF(BARCODE));
	FB_TCP_CLIENT.ENABLE:=FALSE;
	FB_TCP_CLIENT.RESET:=TRUE;
	STATE:=0;
END_IF
FB_CALL_ACT();
CASE STATE OF
	100:
		DONE:=FALSE;
		FB_TCP_CLIENT.RESET:=FALSE;
		FB_TCP_CLIENT.ENABLE:=TRUE;
		MEMSET(ADR(BARCODE),0,SIZEOF(BARCODE));
		IF FB_TCP_CLIENT.CONNECTION_STATE=ESOCKET_CONNECTED THEN
			STATE:=200;
		END_IF
	200:
		IF FB_TCP_CLIENT.SEND(STR_LON, INT_TO_UDINT(LEN(STR_LON)), TCP_BUFF) THEN
			MEMSET(ADR(BARCODE),0,SIZEOF(BARCODE));
			MEMCPY(ADR(BARCODE), ADR(TCP_BUFF), INT_TO_UDINT(LEN(TCP_BUFF)));
			STATE:=300;
		END_IF	
	300:
		DONE:=TRUE;
		FB_TCP_CLIENT.RESET:=FALSE;
		FB_TCP_CLIENT.ENABLE:=FALSE;
		MEMSET(ADR(TCP_BUFF),0,SIZEOF(TCP_BUFF));
		IF FB_TCP_CLIENT.CONNECTION_STATE=ESOCKET_DISCONNECTED THEN
			STATE:=400;
		END_IF
END_CASE

ACTION FB_CALL_ACT:
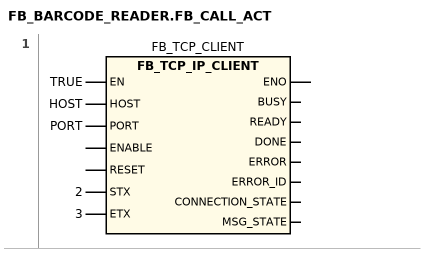
// NETWORK 1
FB_TCP_CLIENT(HOST := HOST, PORT := PORT, STX := 2, ETX := 3); // FB_TCP_IP_CLIENT
END_ACTION

METHOD PUBLIC READ : BOOL
VAR_INPUT
END_VAR
READ:= (STATE=400 OR STATE=9999);
IF NOT READ AND STATE=0 THEN
	STATE:=100;
END_IF
IF READ AND STATE=400 THEN
	STATE:=0;
END_IF
END_METHOD

METHOD PUBLIC READ_REF : BOOL
VAR_INPUT
	pData:				PVOID;
	nData:				UDINT;
END_VAR
READ_REF:= (STATE=400 OR STATE=9999);
IF NOT READ_REF AND STATE=0 THEN
	STATE:=100;
END_IF
IF READ_REF AND STATE=400 THEN
	MEMSET(pData,0,nData);
	MEMCPY(pData, ADR(BARCODE), INT_TO_UDINT(MIN(LEN(BARCODE), UDINT_TO_INT(nData))));
	STATE:=0;
END_IF
END_METHOD

END_FUNCTION_BLOCK

// TcpIpClients/FB_TCP_IP_CLIENT
FUNCTION_BLOCK FB_TCP_IP_CLIENT
VAR_INPUT
	HOST:				T_IPV4ADDR := '';
	PORT:				UDINT;
	ENABLE:				BOOL;
	RESET:				BOOL;
	STX:				BYTE:=DEFAULT_STX;
	ETX:				BYTE:=DEFAULT_ETX;
END_VAR
VAR_OUTPUT
	BUSY:				BOOL;
	READY:				BOOL;
	DONE:				BOOL;
	
	ERROR:				BOOL;
	ERROR_ID:			UDINT;
	
	CONNECTION_STATE:	E_SOCKETCONNECTIONSTATE := ESOCKET_DISCONNECTED;
	MSG_STATE: 			ENUM_DATA_EXCHANGE_STATE := E_IDLE;
END_VAR
VAR
	FB_CLIENT:			FB_ClientServerConnection;
	FB_SEND:			FB_SocketSend;
	FB_RECEIVE:			FB_SocketReceive;
	H_SOCKET:			T_HSOCKET;
	
	TX_BUFF, RX_BUFF:								ARRAY[0..DEFAULT_SDAT_LENGTH+1] OF BYTE;
	RX_BUFF_OUT, TX_BUFF_IN:						STRING[DEFAULT_SDAT_LENGTH];
	
    TON_RCV, TON_DC:								TON;	
   	LEN_REC, LEN_FRAME, START_POS, END_POS, IDX, LEN_MSG:	UDINT;
	STATE:											ENUM_DATA_EXCHANGE_STATE;
	EXECUTE:										BOOL;
	RT_EXECUTE, RT_CONNECTED, RT_DISCONNECTED, RT_RESET:	R_TRIG;
	
	eSubSystem: 			E_SubSystem:= E_SubSystem.LOGIC;
	FB_LOGGER:				FB_EventLogger:= (eSubsystem:= eSubsystem);
END_VAR

MSG_STATE:=STATE;
RT_EXECUTE(CLK:=EXECUTE);
RT_RESET(CLK:=RESET);
RT_CONNECTED(CLK:=CONNECTION_STATE=ESOCKET_CONNECTED);
RT_DISCONNECTED(CLK:=CONNECTION_STATE=ESOCKET_DISCONNECTED);

IF RT_DISCONNECTED.Q THEN
	//FB_LOGGER(sMsg:='Disconnected.', eSevr:=TcEventSeverity.Info);
END_IF
IF RT_CONNECTED.Q THEN
	//FB_LOGGER(sMsg:=CONCAT('Connected to: ', HOST), eSevr:=TcEventSeverity.Info);
END_IF
IF RT_RESET.Q THEN
	//FB_LOGGER(sMsg:=CONCAT('Reseted externaly - ERROR_ID: ', UDINT_TO_STRING(ERROR_ID)), eSevr:=TcEventSeverity.Info);
	FB_SEND.bExecute:=FALSE;
	FB_RECEIVE.bExecute:=FALSE;
	ERROR_ID:= 0;
	STATE:=E_IDLE;
END_IF

BUSY:= STATE <> E_IDLE;
READY:= STATE = E_IDLE;
ERROR:= STATE = E_ERROR;

CASE STATE OF
	E_IDLE:
		IF RT_EXECUTE.Q THEN
			DONE:=FALSE;
			LEN_REC := 0;
			TON_RCV(IN:= FALSE, PT:= T#0S);
			TON_DC(IN:= FALSE, PT:= T#0S);			
			FB_SEND.bExecute:= FALSE;
			TX_BUFF[0]:= STX;
			MEMCPY(ADR(TX_BUFF)+1,ADR(TX_BUFF_IN),SIZEOF(TX_BUFF_IN));
			TX_BUFF[LEN_MSG+1]:= ETX;
			STATE:=E_SEND_START;
		END_IF
	
	E_SEND_START:
		FB_SEND.bExecute:= TRUE;
		STATE:=E_SEND_WAIT;
		
	E_SEND_WAIT:
		FB_SEND.bExecute:= FALSE;
		IF NOT FB_SEND.bBusy THEN
			IF NOT FB_SEND.bError THEN
				STATE:= E_RECEIVE_START;
			ELSE
				ERROR_ID := FB_SEND.nErrId;
				FB_LOGGER(sMsg:=CONCAT('FB_SEND throw an error -  ERROR_ID: ', UDINT_TO_STRING(FB_SEND.nErrId)), eSevr:=TcEventSeverity.Error);
			END_IF
		END_IF
		
	E_RECEIVE_START:
		TON_DC();
		TON_RCV(IN:=TRUE);
		IF TON_RCV.Q THEN
			TON_RCV(IN:= FALSE);
			FB_RECEIVE.bExecute:= TRUE;
			STATE := E_RECEIVE_WAIT;
		END_IF
		
	E_RECEIVE_WAIT:
		FB_RECEIVE.bExecute:= FALSE;
		IF NOT FB_RECEIVE.bBusy THEN
			IF NOT FB_RECEIVE.bError THEN
				 IF FB_RECEIVE.nRecBytes>0 THEN 					(* bytes received *)
					
					START_POS:= LEN_REC;							(* rxBuffer array index of first data byte *)
					END_POS:= LEN_REC + FB_RECEIVE.nRecBytes - 1;	(* rxBuffer array index of last data byte *)
					LEN_REC:= LEN_REC + FB_RECEIVE.nRecBytes;		(* calculate the number of received data bytes *)
					LEN_FRAME:= 0;									(* reset frame length *)
					
					IF LEN_REC < SIZEOF(RX_BUFF_OUT) THEN			(* no overflow *)
						TON_RCV(PT:= T#0S); 						(* bytes received => increase the read (polling) speed *)
						TON_DC(IN := FALSE);						(* bytes received => disable timeout check *)
						
						(* search for string end delimiter *)
						FOR idx := START_POS TO END_POS BY 1 DO
							IF RX_BUFF[IDX] = 16#00 THEN												(* string end delimiter found *)
								LEN_FRAME := IDX + 1;													(* calculate the length of the received string (inclusive the end delimiter) *)
								MEMCPY(ADR(RX_BUFF_OUT), ADR(RX_BUFF), LEN_FRAME );						(* copy the received string to the output variable (inclusive the end delimiter) *)
								MEMMOVE( ADR(RX_BUFF), ADR(RX_BUFF[LEN_FRAME]), LEN_REC-LEN_FRAME );	(* move the reamaining data bytes *)
								//ADSLOGSTR( ADSLOG_MSGTYPE_HINT OR ADSLOG_MSGTYPE_LOG, 'RX_BUFF_OUT: %s', RX_BUFF_OUT );
								LEN_REC:= LEN_REC-LEN_FRAME;											(* recalculate the remaining data byte length *)
								STATE:= E_DONE;
								EXIT;
							END_IF
						END_FOR					
					ELSE						(* there is no more free read buffer space => the answer string should be terminated *)
						ERROR_ID:= 15001;		(* buffer overflow !*)
						FB_LOGGER(sMsg:=CONCAT('Buffer overflow error, the recived data size is bigger than the RxBuffer. - ERROR_ID: ', UDINT_TO_STRING(ERROR_ID)), eSevr:=TcEventSeverity.Error);
					END_IF				
				ELSE										(* no bytes received *)
					TON_RCV(PT:= T#100MS);					(* no bytes received => decrease the read (polling) speed *)
					TON_DC(IN:= TRUE, PT:= T#10S);			(* no bytes received => enable timeout check*)
					IF TON_DC.Q THEN 						(* timeout error*)
						TON_DC(IN:= FALSE);					
						ERROR_ID:= 15002;
						FB_LOGGER(sMsg:=CONCAT('Timeout error, T#10s response timer is elapsed. - ERROR_ID: ', UDINT_TO_STRING(ERROR_ID)), eSevr:=TcEventSeverity.Error);
					ELSE							(* repeat reading *)
						STATE:= E_RECEIVE_START;
					END_IF
				END_IF
			ELSE									(* receive error *)
				ERROR_ID := FB_RECEIVE.nErrId;
				FB_LOGGER(sMsg:=CONCAT('FB_RECEIVE throw an error -  ERROR_ID: ', UDINT_TO_STRING(FB_RECEIVE.nErrId)), eSevr:=TcEventSeverity.Error);
			END_IF
		   END_IF		
	
	E_DONE:
		DONE:=TRUE;
		IF NOT EXECUTE THEN
			LEN_REC:=0;
			FB_SEND.bExecute:=FALSE;
			FB_RECEIVE.bExecute:=FALSE;
			STATE:= E_IDLE;
		END_IF
		
	E_ERROR:
		DONE:=TRUE;
		IF NOT EXECUTE THEN
			LEN_REC:=0;
			FB_SEND.bExecute:=FALSE;
			FB_RECEIVE.bExecute:=FALSE;
			ERROR_ID:=0;
			STATE:= E_IDLE;
		END_IF
		
END_CASE

IF ERROR_ID <> 0 THEN
	STATE:= E_ERROR;
END_IF

FB_CALL_ACT();

ACTION FB_CALL_ACT:
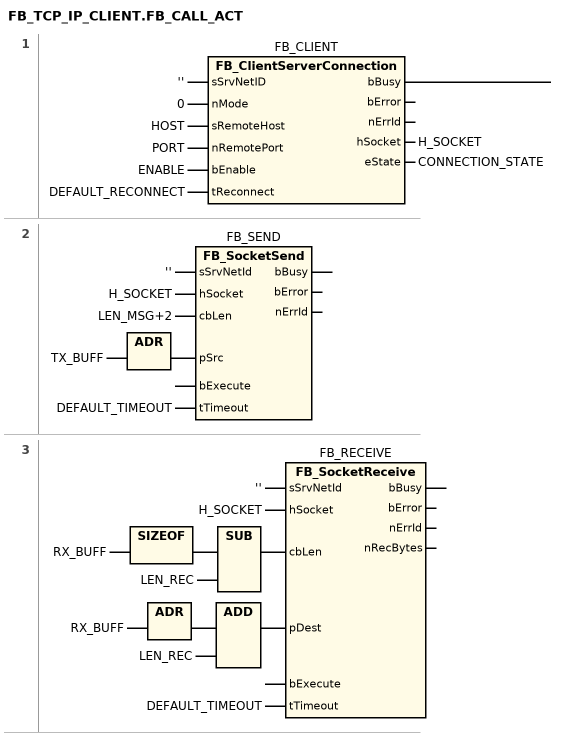
// NETWORK 1
FB_CLIENT(
    sSrvNetID := '',
    nMode := 0,
    sRemoteHost := HOST,
    nRemotePort := PORT,
    bEnable := ENABLE,
    tReconnect := DEFAULT_RECONNECT,
    hSocket => H_SOCKET,
    eState => CONNECTION_STATE); // FB_ClientServerConnection

// NETWORK 2
FB_SEND(
    sSrvNetId := '',
    hSocket := H_SOCKET,
    cbLen := LEN_MSG+2,
    pSrc := ADR(TX_BUFF),
    tTimeout := DEFAULT_TIMEOUT); // FB_SocketSend

// NETWORK 3
FB_RECEIVE(
    sSrvNetId := '',
    hSocket := H_SOCKET,
    cbLen := SIZEOF(RX_BUFF) - LEN_REC,
    pDest := ADR(RX_BUFF) + LEN_REC,
    tTimeout := DEFAULT_TIMEOUT); // FB_SocketReceive
END_ACTION

METHOD PUBLIC SEND : BOOL
VAR_INPUT
	MESSAGE:		REFERENCE TO STRING[DEFAULT_SDAT_LENGTH];
	MSG_LENGTH:		UDINT;
	RECIVED:		REFERENCE TO STRING[DEFAULT_SDAT_LENGTH];
END_VAR
IF STATE= E_IDLE THEN
	LEN_MSG:=MSG_LENGTH;
	TX_BUFF_IN:= MESSAGE;
	EXECUTE:=TRUE;
	SEND:=FALSE;
END_IF

IF STATE= E_DONE THEN
	RECIVED:= RX_BUFF_OUT;	
	EXECUTE:=FALSE;
	SEND:=TRUE;
END_IF
IF STATE= E_ERROR THEN
	RECIVED:= 'ERROR';	
	EXECUTE:=FALSE;
	SEND:=TRUE;
END_IF
END_METHOD

END_FUNCTION_BLOCK

// TcpIpClients/FB_TCP_IP_CLIENT_LDAT
FUNCTION_BLOCK FB_TCP_IP_CLIENT_LDAT
VAR_INPUT
	HOST:				T_IPV4ADDR := '';
	PORT:				UDINT;
	ENABLE:				BOOL;
	RESET:				BOOL;
	STX:				BYTE:=DEFAULT_STX;
	ETX:				BYTE:=DEFAULT_ETX;
END_VAR
VAR_OUTPUT
	BUSY:				BOOL;
	READY:				BOOL;
	DONE:				BOOL;
	
	ERROR:				BOOL;
	ERROR_ID:			UDINT;
	
	CONNECTION_STATE:	E_SOCKETCONNECTIONSTATE := ESOCKET_DISCONNECTED;
	MSG_STATE: 			ENUM_DATA_EXCHANGE_STATE := E_IDLE;
END_VAR
VAR
	FB_CLIENT:			FB_ClientServerConnection;
	FB_SEND:			FB_SocketSend;
	FB_RECEIVE:			FB_SocketReceive;
	H_SOCKET:			T_HSOCKET;
	
	TX_BUFF, RX_BUFF:								ARRAY[0..DEFAULT_LDAT_LENGTH+1] OF BYTE;
	RX_BUFF_OUT, TX_BUFF_IN:						STRING[DEFAULT_LDAT_LENGTH];
	
    TON_RCV, TON_DC:								TON;	
   	LEN_REC, LEN_FRAME, START_POS, END_POS, IDX, LEN_MSG:	UDINT;
	STATE:											ENUM_DATA_EXCHANGE_STATE;
	EXECUTE:										BOOL;
	RT_EXECUTE, RT_CONNECTED, RT_DISCONNECTED, RT_RESET:	R_TRIG;
	
	eSubSystem: 			E_SubSystem:= E_SubSystem.LOGIC;
	FB_LOGGER:				FB_EventLogger:= (eSubsystem:= eSubsystem);
END_VAR

MSG_STATE:=STATE;
RT_EXECUTE(CLK:=EXECUTE);
RT_RESET(CLK:=RESET);
RT_CONNECTED(CLK:=CONNECTION_STATE=ESOCKET_CONNECTED);
RT_DISCONNECTED(CLK:=CONNECTION_STATE=ESOCKET_DISCONNECTED);

IF RT_DISCONNECTED.Q THEN
	//FB_LOGGER(sMsg:='Disconnected.', eSevr:=TcEventSeverity.Info);
END_IF
IF RT_CONNECTED.Q THEN
	//FB_LOGGER(sMsg:=CONCAT('Connected to: ', HOST), eSevr:=TcEventSeverity.Info);
END_IF
IF RT_RESET.Q THEN
	//FB_LOGGER(sMsg:=CONCAT('Reseted externaly - ERROR_ID: ', UDINT_TO_STRING(ERROR_ID)), eSevr:=TcEventSeverity.Info);
	FB_SEND.bExecute:=FALSE;
	FB_RECEIVE.bExecute:=FALSE;
	ERROR_ID:= 0;
	STATE:=E_IDLE;
END_IF

BUSY:= STATE <> E_IDLE;
READY:= STATE = E_IDLE;
ERROR:= STATE = E_ERROR;

CASE STATE OF
	E_IDLE:
		IF RT_EXECUTE.Q THEN
			ERROR_ID:=0;
			DONE:=FALSE;
			LEN_REC := 0;
			TON_RCV(IN:= FALSE, PT:= T#0S);
			TON_DC(IN:= FALSE, PT:= T#0S);			
			FB_SEND.bExecute:= FALSE;
			TX_BUFF[0]:= STX;
			MEMCPY(ADR(TX_BUFF)+1,ADR(TX_BUFF_IN),SIZEOF(TX_BUFF_IN));
			TX_BUFF[LEN_MSG]:= ETX;
			LEN_MSG:=LEN_MSG+1;
			STATE:=E_SEND_START;
		END_IF
	
	E_SEND_START:
		FB_SEND.bExecute:= TRUE;
		STATE:=E_SEND_WAIT;
		
	E_SEND_WAIT:
		FB_SEND.bExecute:= FALSE;
		IF NOT FB_SEND.bBusy THEN
			IF NOT FB_SEND.bError THEN
				STATE:= E_RECEIVE_START;
			ELSE
				ERROR_ID := FB_SEND.nErrId;
				FB_LOGGER(sMsg:=CONCAT('FB_SEND throw an error -  ERROR_ID: ', UDINT_TO_STRING(FB_SEND.nErrId)), eSevr:=TcEventSeverity.Error);
			END_IF
		END_IF
		
	E_RECEIVE_START:
		TON_DC();
		TON_RCV(IN:=TRUE);
		IF TON_RCV.Q THEN
			TON_RCV(IN:= FALSE);
			FB_RECEIVE.bExecute:= TRUE;
			STATE := E_RECEIVE_WAIT;
		END_IF
		
	E_RECEIVE_WAIT:
		FB_RECEIVE.bExecute:= FALSE;
		IF NOT FB_RECEIVE.bBusy THEN
			IF NOT FB_RECEIVE.bError THEN
				 IF FB_RECEIVE.nRecBytes>0 THEN 					(* bytes received *)
					
					START_POS:= LEN_REC;							(* rxBuffer array index of first data byte *)
					END_POS:= LEN_REC + FB_RECEIVE.nRecBytes - 1;	(* rxBuffer array index of last data byte *)
					LEN_REC:= LEN_REC + FB_RECEIVE.nRecBytes;		(* calculate the number of received data bytes *)
					LEN_FRAME:= 0;									(* reset frame length *)
					
					IF LEN_REC < SIZEOF(RX_BUFF_OUT) THEN			(* no overflow *)
						TON_RCV(PT:= T#0S); 						(* bytes received => increase the read (polling) speed *)
						TON_DC(IN := FALSE);						(* bytes received => disable timeout check *)
						
						(* search for string end delimiter *)
						FOR idx := START_POS TO END_POS BY 1 DO
							IF RX_BUFF[IDX] = 16#00 THEN												(* string end delimiter found *)
								LEN_FRAME := IDX + 1;													(* calculate the length of the received string (inclusive the end delimiter) *)
								MEMCPY(ADR(RX_BUFF_OUT), ADR(RX_BUFF), LEN_FRAME );						(* copy the received string to the output variable (inclusive the end delimiter) *)
								MEMMOVE( ADR(RX_BUFF), ADR(RX_BUFF[LEN_FRAME]), LEN_REC-LEN_FRAME );	(* move the reamaining data bytes *)
								LEN_REC:= LEN_REC-LEN_FRAME;											(* recalculate the remaining data byte length *)
								STATE:= E_DONE;
								EXIT;
							END_IF
						END_FOR					
					ELSE						(* there is no more free read buffer space => the answer string should be terminated *)
						ERROR_ID:= 15001;		(* buffer overflow !*)
						FB_LOGGER(sMsg:=CONCAT('Buffer overflow error, the recived data size is bigger than the RxBuffer. - ERROR_ID: ', UDINT_TO_STRING(ERROR_ID)), eSevr:=TcEventSeverity.Error);
					END_IF				
				ELSE										(* no bytes received *)
					TON_RCV(PT:= T#100MS);					(* no bytes received => decrease the read (polling) speed *)
					TON_DC(IN:= TRUE, PT:= T#10S);			(* no bytes received => enable timeout check*)
					IF TON_DC.Q THEN 						(* timeout error*)
						TON_DC(IN:= FALSE);					
						ERROR_ID:= 15002;
						FB_LOGGER(sMsg:=CONCAT('Timeout error, T#10s response timer is elapsed. - ERROR_ID: ', UDINT_TO_STRING(ERROR_ID)), eSevr:=TcEventSeverity.Error);
					ELSE							(* repeat reading *)
						STATE:= E_RECEIVE_START;
					END_IF
				END_IF
			ELSE									(* receive error *)
				ERROR_ID := FB_RECEIVE.nErrId;
				FB_LOGGER(sMsg:=CONCAT('FB_RECEIVE throw an error -  ERROR_ID: ', UDINT_TO_STRING(FB_RECEIVE.nErrId)), eSevr:=TcEventSeverity.Error);
			END_IF
		   END_IF		
	
	E_DONE:
		DONE:=TRUE;
		IF NOT EXECUTE THEN
			LEN_REC:=0;
			FB_SEND.bExecute:=FALSE;
			FB_RECEIVE.bExecute:=FALSE;
			STATE:= E_IDLE;
		END_IF
		
	E_ERROR:
		DONE:=TRUE;
		IF NOT EXECUTE THEN
			LEN_REC:=0;
			FB_SEND.bExecute:=FALSE;
			FB_RECEIVE.bExecute:=FALSE;
			//ERROR_ID:=0;
			STATE:= E_IDLE;
		END_IF
		
END_CASE

IF ERROR_ID <> 0 THEN
	STATE:= E_ERROR;
END_IF

FB_CALL_ACT();

ACTION FB_CALL_ACT:
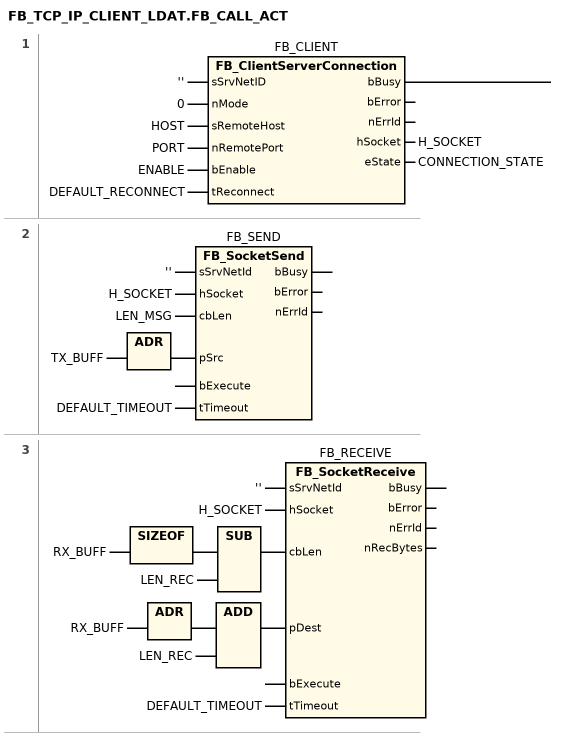
// NETWORK 1
FB_CLIENT(
    sSrvNetID := '',
    nMode := 0,
    sRemoteHost := HOST,
    nRemotePort := PORT,
    bEnable := ENABLE,
    tReconnect := DEFAULT_RECONNECT,
    hSocket => H_SOCKET,
    eState => CONNECTION_STATE); // FB_ClientServerConnection

// NETWORK 2
FB_SEND(
    sSrvNetId := '',
    hSocket := H_SOCKET,
    cbLen := LEN_MSG,
    pSrc := ADR(TX_BUFF),
    tTimeout := DEFAULT_TIMEOUT); // FB_SocketSend

// NETWORK 3
FB_RECEIVE(
    sSrvNetId := '',
    hSocket := H_SOCKET,
    cbLen := SIZEOF(RX_BUFF) - LEN_REC,
    pDest := ADR(RX_BUFF) + LEN_REC,
    tTimeout := DEFAULT_TIMEOUT); // FB_SocketReceive
END_ACTION

METHOD PUBLIC SEND : BOOL
VAR_INPUT
	MESSAGE:		REFERENCE TO STRING[DEFAULT_LDAT_LENGTH];
	MSG_LENGTH:		UDINT;
	RECIVED:		REFERENCE TO STRING[DEFAULT_LDAT_LENGTH];
END_VAR
IF STATE= E_IDLE THEN
	LEN_MSG:=MSG_LENGTH;
	TX_BUFF_IN:= MESSAGE;
	EXECUTE:=TRUE;
	SEND:=FALSE;
END_IF

IF STATE= E_DONE THEN
	RECIVED:= RX_BUFF_OUT;	
	EXECUTE:=FALSE;
	SEND:=TRUE;
END_IF
IF STATE= E_ERROR THEN
	RECIVED:= 'ERROR';	
	EXECUTE:=FALSE;
	SEND:=TRUE;
END_IF
END_METHOD

END_FUNCTION_BLOCK

// Test/MAIN
PROGRAM MAIN
VAR

END_VAR

ACTION FB_CALL_ACT:

END_ACTION

END_PROGRAM
